   #mb_query.mode := #mb_query.c.mode.write;
   #mb_query(data_addr := 40060, data_ptr := #setting);

   "mb_station_block_footer"(sb := #sb, mb_query := #mb_query);

   (*
   Setting:

   value[1] and value[2]
   ------------------
   2 = Pascal (Pa)
   3 = kiloPascal (kPa)
   4 = megaPascal (MPa)
   5 = pounds per square inch (psi)
   6 = inches of water at 68 F
   7 = ftH2O
   8 = atm
   9 = bar
   10 = kg/cm2
   11 = g/cm2
   12 = cmHg
   13 = mmHg
   14 = torr
   15 = mH2O
   16 = cmH2O
   17 = mmH2O
   18 = inHg
   19 = mbar


   value[3]
   ------------------
   20 = degrees Celsius (ï‚°C)
   21 = degrees Fahrenheit (ï‚°F)
   22 = degrees Kelvin (K)
   23 = degrees Rankine(R)

   *)
END_FUNCTION_BLOCK

FUNCTION_BLOCK "Schneider_conzerv_EM6430"   // FB91, SCL
{ S7_Optimized_Access := 'TRUE' }
VERSION : 0.1
   VAR_INPUT
      mb_addr : USInt;
   END_VAR
   VAR_IN_OUT
      mb_query : "mb_query";
   END_VAR
   VAR
      sb : "mb_station_block_udt";
      read1_common : Struct
         Apparent_power_total : Real;
         Active_power_total : Real;
         Reactive_power_total : Real;
         Power_factor_average : Real;
         Voltage_average_phase_phase : Real;
         Voltage_average_phase_neutral : Real;
         Current_average : Real;
         Frequency : Real;   // Hz
      END_STRUCT;
      read2_phase : Array[1..3] of Struct
         Apparent_power : Real;
         Active_power : Real;
         Reactive_power : Real;
         Power_factor : Real;
         Voltage_phase_phase : Real;
         Voltage_phase_neutral : Real;
         Current : Real;
      END_STRUCT;
      read3_THD : Struct
         Voltage_THD : Array[1..3] of Real;
         Current_THD : Array[1..3] of Real;
      END_STRUCT;
      read4 : Struct
         Forward_apparent_energy : Real;
         Forward_active_energy : Real;
         Forward_reactive_inductive_energy : Real;
         Forward_reactive_capacitive_energy : Real;
         Reverse_apparent_energy : Real;
         Reverse_active_energy : Real;
         Reverse_reactive_inductive_Energy : Real;
         Reverse_reactive_capacitive_Energy : Real;
         Average_load_percentage : Real;
         Percentage_of_phase_load : Array[1..3] of Real;
         "Unbalanced_%load" : Real;
         "Unbalanced_%_voltage" : Real;
      END_STRUCT;
      read5_common_RMS : Struct
         Apparent_power_total : Real;
         Active_power_total : Real;
         Reactive_power_total : Real;
         Power_factor_average : Real;
         Voltage_average_phase_phase : Real;
         Voltage_average_phase_neutral : Real;
         Current_average : Real;
         Frequency : Real;   // Hz
         _ : UDInt;   // Reserved
         Number_of_interruption : UDInt;
      END_STRUCT;
   END_VAR
BEGIN
   // Schneider-electric - Conzerv EM6430 - Power meters
   // NHA12535-03
   // 
   // https://www.schneider-electric.com/resources/sites/SCHNEIDER_ELECTRIC/
   // content/live/FAQS/276000/FA276938/en_US/EM6430_User_Manual_NHA12535-03.pdf

   "mb_station_block_header"(sb := #sb, mb_query := #mb_query);
   #mb_query.mb_addr := #mb_addr; // Device address.

   #mb_query.mode := #mb_query.c.read.holding_reg;
   #mb_query(data_addr := 3901, data_ptr := #read1_common);
   #mb_query(data_addr := 3917, data_ptr := #read2_phase);
   #mb_query(data_addr := 3861, data_ptr := #read3_THD);
   #mb_query(data_addr := 3959, data_ptr := #read4);
   #mb_query(data_addr := 3001, data_ptr := #read5_common_RMS);

   "mb_station_block_footer"(sb := #sb, mb_query := #mb_query);
END_FUNCTION_BLOCK

// folder: Library/Modbus/Station blocks/sb Untested/S/Schneider/Altivar

FUNCTION_BLOCK "Schneider_Altivar_21_simple"   // FB123, SCL
{ S7_Optimized_Access := 'TRUE' }
VERSION : 0.1
   VAR_INPUT
      mb_addr : UInt;
      ref : Real;   // Percent
   END_VAR
   VAR_OUTPUT
      Output_frequency : Real;
   END_VAR
   VAR_IN_OUT
      mb_query : "mb_query";
   END_VAR
   VAR
      sb : "mb_station_block_udt";
      read : Struct   // 16#fd00
         frequency : Word;
         stat : Struct
            x08 : Bool;
            x09_Reverse : Bool;
            x10_Run : Bool;
            x11_Coast_stop : Bool;
            x12_Emergency_stop : Bool;
            x13_Standby_ST_ON : Bool;   // Standby: Initialization completed, not failure stop status, not alarm stop status (MOFF, LL forced stop or forced stop due to a momentary power failure), ST=ON, and RUN=ON
            x14_Standby : Bool;   // Standby: Initialization completed, not failure stop status, and not alarm stop status (MOFF, LL forced stop or forced stop due to a momentary power failure)
            x15_Local : Bool;
            x00_Failure_FL : Bool;
            x01_Failure : Bool;
            x02_Alarm : Bool;
            x03_Main_circuit_undervoltage : Bool;
            x04_THR_2 : Bool;   // THR1: PT=set value, vL, vb, Thr - THR2: PT=0, F170, F172, F173
            x05_PI_control_OFF : Bool;
            x06_Acceleration2_deceleration2 : Bool;
            x07_DC_braking : Bool;
         END_STRUCT;
      END_STRUCT;
      write : Struct
         cmd : Struct
            x08 : Bool;   // [08]
            reverse : Bool;   // [09]
            run : Bool;   // [10]
            coast_stop : Bool;   // [11]
            emergency_stop : Bool;   // [12]
            fault_reset : Bool;   // [13]
            setpoint_priority : Bool := TRUE;   // [14] Enabled regardless of the setting of FMOD
            command_priority : Bool := TRUE;   // [15] Enabled regardless of the setting of CMOD
            preset_speed_b0 : Bool;   // [00]
            preset_speed_b1 : Bool;   // [01]
            preset_speed_b2 : Bool;   // [02]
            x03 : Bool;   // [03]
            thr2 : Bool;   // [04] THR1 : PT=set value, vL, vb, tHr - THR2 : PT=0, F170, F172, F173
            PI_control : Bool;   // [05] 0:Normal operation, 1:PI OFF
            acceleration_deceleration_pattern_2 : Bool;   // [06] 0: Acceleration deceleration pattern 1
            DC_braking : Bool;   // [07]
         END_STRUCT;
         ref_speed : UInt;
      END_STRUCT;
   END_VAR
BEGIN
   // Schneider (Telemecanique) - Altivar 21 inverter
   // VFD (AC-drive)

   (*
   Param:  Name:             Default:    Options:          
   F800    Baud rate         19200       0: 9600 bps, 1: 19200 bps     
   F801    Parity            Even        0: None, 1: Even, 2: Odd      
   F802    Modbus address    1           0 ... 247                     

   CMOD    2 -> Serial communication
   FMOD    4 -> Serial communication
   *)

   "mb_station_block_header"(sb := #sb, mb_query := #mb_query);
   #mb_query.mb_addr := #mb_addr;

   #write.ref_speed := REAL_TO_UINT(#ref * 100);
   #write.cmd.run := #ref <> 0;
   #mb_query(mode := #mb_query.c.write.holding_reg,
             data_addr := 16#fa00,
             data_ptr := #write);

   // Basic data, status word.
   #mb_query(mode := #mb_query.c.read.holding_reg,
             data_addr := 16#fd00,
             data_ptr := #read);
   #Output_frequency := UINT_TO_REAL(#read.frequency) / 100; // [%]

   "mb_station_block_footer"(sb := #sb, mb_query := #mb_query);
END_FUNCTION_BLOCK

// folder: Library/Modbus/Station blocks/sb Untested/S/Schneider/Altivar/Advanced

FUNCTION_BLOCK "Schneider_Altivar_21"   // FB95, SCL
{ S7_Optimized_Access := 'TRUE' }
VERSION : 0.1
   VAR_INPUT
      mb_addr : UInt;
      ref : Real;
      acceleration_time : Real;
   END_VAR
   VAR_IN_OUT
      mb_query : "mb_query";
   END_VAR
   VAR
      sb : "mb_station_block_udt";
      data6 : Struct
         Output_current : Real;
         Voltage_DC_bus : Real;
         Output_frequency : Real;
      END_STRUCT;
      read1 : Struct   // 16#fd00
         Output_frequency : Word;
         stat : Struct
            x08 : Bool;
            x09_Reverse : Bool;
            x10_Run : Bool;
            x11_Coast_stop : Bool;
            x12_Emergency_stop : Bool;
            x13_Standby_ST_ON : Bool;   // Standby: Initialization completed, not failure stop status, not alarm stop status (MOFF, LL forced stop or forced stop due to a momentary power failure), ST=ON, and RUN=ON
            x14_Standby : Bool;   // Standby: Initialization completed, not failure stop status, and not alarm stop status (MOFF, LL forced stop or forced stop due to a momentary power failure)
            x15_Local : Bool;
            x00_Failure_FL : Bool;
            x01_Failure : Bool;
            x02_Alarm : Bool;
            x03_Main_circuit_undervoltage : Bool;
            x04_THR_2 : Bool;   // THR1: PT=set value, vL, vb, Thr - THR2: PT=0, F170, F172, F173
            x05_PI_control_OFF : Bool;
            x06_Acceleration2_deceleration2 : Bool;
            x07_DC_braking : Bool;
         END_STRUCT;
      END_STRUCT;
      read2 : Struct   // 16#fe45
         Command_mode : UInt;   // 0:Terminal board, 1:Operation panel, 2:Serial
         Setpoint_mode : UInt;   // 1 VIA, 2 VIB, 3 Operation panel, 4 Serial, 5 TB up down frequency, 255 Preset speed operation
      END_STRUCT;
      read3_alarm : Struct   // 16#fe91
         x08_Over_torque : Bool;
         x09_Cumulative_operation_hours : Bool;
         x10 : Bool;
         x11 : Bool;
         x12 : Bool;
         "x13_Main circuit_undervoltage" : Bool;   // same as MS-relay status
         x14_Decelerating_stopping : Bool;   // Related: F256 setting. At the time of the instant blackout, Forced deceleration/stop
         x15_Decelerating_stopping : Bool;   // Related: F302 setting. An automatic stop during the lower limit frequency continuance
         x00_Overcurrent : Bool;
         x01_Inverter_overload : Bool;
         x02_Motor_overload : Bool;
         x03_Overheat : Bool;
         x04_Overvoltage : Bool;
         x05_Main_circuit_undervoltage : Bool;
         x06 : Bool;
         x07_Undercurrent : Bool;
      END_STRUCT;
      read4_alarm2 : Struct   // 16#fe79
         x08 : Bool;
         x09 : Bool;
         x10 : Bool;
         x11 : Bool;
         x12 : Bool;
         x13 : Bool;
         x14 : Bool;
         x15 : Bool;
         x00_Fan_life_alarm : Bool;
         x01_Circuit_board_life : Bool;
         x02_Main_circuit_capacitor_life : Bool;
         x03_User_set_alarm : Bool;
         x04 : Bool;
         x05 : Bool;
         x06 : Bool;
         x07 : Bool;
      END_STRUCT;
      read5_trip_code : UInt;   // 16#fc90
      write1 : Struct
         cmd : Struct
            x08 : Bool;   // [08]
            reverse : Bool;   // [09]
            run : Bool;   // [10]
            coast_stop : Bool;   // [11]
            emergency_stop : Bool;   // [12]
            fault_reset : Bool;   // [13]
            setpoint_priority : Bool := TRUE;   // [14] Enabled regardless of the setting of FMOD
            command_priority : Bool := TRUE;   // [15] Enabled regardless of the setting of CMOD
            preset_speed_b0 : Bool;   // [00]
            preset_speed_b1 : Bool;   // [01]
            preset_speed_b2 : Bool;   // [02]
            x03 : Bool;   // [03]
            thr2 : Bool;   // [04] THR1 : PT=set value, vL, vb, tHr - THR2 : PT=0, F170, F172, F173
            PI_control : Bool;   // [05] 0:Normal operation, 1:PI OFF
            acceleration_deceleration_pattern_2 : Bool;   // [06] 0: Acceleration deceleration pattern 1
            DC_braking : Bool;   // [07]
         END_STRUCT;
         ref : UInt;
      END_STRUCT;
      write2_comm_fault_action : UInt;
      _ : Bool;
      sequence : "mb_sequence";
   END_VAR
   VAR_TEMP
      read6 : Struct   // 16#fe03
         Output_current : UInt;
         Voltage_DC_bus : UInt;
      END_STRUCT;
      u : UInt;
   END_VAR
BEGIN
   // Schneider (Telemecanique) - Altivar 21 inverter
   // VFD (AC-drive)

   (*
   Param:  Name:             Default:    Options:          
   F800    Baud rate         19200       0: 9600 bps, 1: 19200 bps     
   F801    Parity            Even        0: None, 1: Even, 2: Odd      
   F802    Modbus address    1           0 ... 247                     

   CMOD    2 -> Serial communication
   FMOD    4 -> Serial communication
   *)

   "mb_station_block_header"(sb := #sb, mb_query := #mb_query);
   #mb_query.mb_addr := #mb_addr;

   REGION Low priority queries     
       #sequence.conf.first_state := 1600;
       CASE "mb_sequence_init"(sequence := #sequence, mb_query := #mb_query) OF
               // ----- READ HOLDING REG ----- (State 3xx)
           300: // Where the drive take commands from: modbus or Terminal board.
               #mb_query(data_addr := 16#fe45, data_ptr := #read2); // 65093
           301: #mb_query(data_addr := 16#fe91, data_ptr := #read3_alarm);
           302: #mb_query(data_addr := 16#fe79, data_ptr := #read4_alarm2);
           303: #mb_query(data_addr := 16#fc90, data_ptr := #read5_trip_code);
           304: // Other data: Current, DC-bus
               #mb_query(data_addr := 16#fe03, data_ptr := #read6);
               IF #mb_query.Done THEN
                   #data6.Output_current := UINT_TO_REAL(#read6.Output_current) / 100;
                   #data6.Voltage_DC_bus := UINT_TO_REAL(#read6.Voltage_DC_bus) / 100;
               END_IF;
               #sequence.next_state := 1600;

               // ----- WRITE MULTIPLE HOLDING REG ----- (State 16xx)
           1600: // Behaviour on modbus fault
               #mb_query(data_addr := 16#f603, data_ptr := #write2_comm_fault_action);
           1601: // Acceleration time 1  (0.1)
               #u := REAL_TO_UINT(#acceleration_time * 10);
               #mb_query(data_addr := 16#f603, data_ptr := #u);
               #sequence.next_state := 300;
           ELSE
               #sequence.state += 1;
       END_CASE;
       #sequence(sb := #sb, mb_query := #mb_query);
   END_REGION

   REGION High priotiry querie     
       #write1.ref := REAL_TO_UINT(#ref * 100);
       #write1.cmd.run := #ref <> 0 AND #sequence.Done;
       #mb_query(mode := #mb_query.c.write.holding_reg, // 64000
                 data_addr := 16#fa00,
                 data_ptr := #write1);

       // Basic data, status word.
       #mb_query(mode := #mb_query.c.read.holding_reg,
                 data_addr := 16#fd00,
                 data_ptr := #read1); // 64768
       IF #mb_query.Done THEN
           #data6.Output_frequency :=
           (* *)UINT_TO_REAL(#read1.Output_frequency) / 100; // [%]
       END_IF;
   END_REGION

   "mb_station_block_footer"(sb := #sb, mb_query := #mb_query);

   (* Trip codes:
   NErr     0  0  No error
   OC1      1  1  Over-current during acceleration
   OC2      2  2  Over-current during deceleration
   OC3      3  3  Over-current during constant speed operation
   OCL      4  4  Over-current in load at startup
   OCA      5  5  Short circuit in arm
   EPHI     8  8  Input phase failure
   EPHO     9  9  Output phase failure
   OP1      A 10 Overvoltage during acceleration
   OP2      B 11 Overvoltage during deceleration
   OP3      C 12 Overvoltage during constant speed operation
   OL1      D 13 Over-LOAD in inverter
   OL2      E 14 Over-LOAD in motor
   OH      10 16 Overheat trip
   E       11 17 Emergency stop
   EEP1    12 18 EEPROM fault 1 (writing error)
   EEP2    13 19 EEPROM fault 2 (reading error)
   EEP3    14 20 EEPROM fault 3 (internal fault)
   Err2    15 21 RAM fault
   Err3    16 22 ROM fault
   Err4    17 23 CPU fault
   Err5    18 24 Communication error trip
   Err7    1A 26 Current detector fault
   Err8    1B 27 Optional circuit board type error
   UC      1D 29 Small-current trip
   UP1     1E 30 Trip due to undervoltage in main circuit
   Ot      20 32 Over-torque trip
   EF2     22 34 Ground fault trip (hardware detection)
   OC1P    25 37 Overcurrent flowing in element during acceleration
   OC2P    26 38 Overcurrent flowing in element during deceleration
   OC3P    27 39 Overcurrent flowing in element during operation
   EtYP    29 41 Inverter type error
   OH2     2E 46 External thermal input
   SOUt    2F 47 VIA cable break
   E-18    32 50 Break in an analog signal cable
   E-19    33 51 CPU fault
   E-20    34 52 Excess torque boost
   E-21    35 53 CPU fault
   Etn1    54 84 Auto-tuning error
   *)
END_FUNCTION_BLOCK

// folder: Library/Modbus/Station blocks/sb Untested/S/Schneider/Power meters

FUNCTION_BLOCK "Schneider_power_meter"   // FB2, SCL
{ S7_Optimized_Access := 'TRUE' }
VERSION : 0.1
   VAR_INPUT
      mb_addr : USInt;
   END_VAR
   VAR_IN_OUT
      mb_query : "mb_query";
   END_VAR
   VAR RETAIN
      conf : Struct
         power_system : UInt := 65535;   // 0=1PH2W L–N, 1=1PH2W L–L, 2=1PH3W L–L with N, 3=3PH3W, 11=3PH4W, 13=1PH4W multi-L with N
      END_STRUCT;
   END_VAR
   VAR
      sb : "mb_station_block_udt";
      "e" : Int;   // Error
      data : "energy_udt";
      frequency : Real;
      temperature : Real;
      serial_number : UDInt;
      power_factor : Struct
         L : Array[1..3] of Real;
         total : Real;
         displacement : Struct
            L : Array[1..3] of Real;
            total : Real;
         END_STRUCT;
      END_STRUCT;
      unbalanced : Struct
         current : Struct
            L : Array[1..3] of Real;
            worst : Real;
         END_STRUCT;
         voltage : Struct
            L_L : Array[1..3] of Real;
            L_L_worst : Real;
            L_N : Array[1..3] of Real;
            L_N_worst : Real;
         END_STRUCT;
      END_STRUCT;
      tangent_phi : Real;
      tmp : DWord;
   END_VAR
   VAR CONSTANT
      ALL : DInt := 0;
   END_VAR
BEGIN
   // Schneider - PowerLogic  (Power meter)
   // PM3200, PM3210, PM3250, PM3255, PM5560, PM5563, PM5563RD
   //
   // DOCA0006EN-06  -  08/2016
   // Default com.: 19200/8-E-1. Default addr: 1
   // 
   // https://www.se.com/ww/en/product/METSEPM3250/pm3250-power-meter---rs485/
   // https://download.schneider-electric.com/files?p_enDocType=User+guide&p_File_Name=DOCA0006EN-06.pdf&p_Doc_Ref=DOCA0006EN
   // https://www.schneider-electric.com/en/faqs/FA234017/
   //
   // Apparently there is a error in the datasheet, all register
   // addresses are added by two. Eg 3000 is actually 2998.

   "mb_station_block_header"(sb := #sb, mb_query := #mb_query );
   #mb_query.mb_addr := #mb_addr;
   #mb_query.mode := #mb_query.c.read.holding_reg;

   IF "mb_query_range"(start := 128, end := 129, q := #mb_query) THEN
       #"e" += "mb_swap_word"(start := #ALL, end := #ALL,  q := #mb_query);
       #"e" += "mb_read_buffer"(addr := 130-2, ptr := #serial_number, q := #mb_query);
   END_IF;

   IF "mb_query_range"(start := 2700-2, end := 2710-1, q := #mb_query) THEN
       #"e" += "mb_swap_word"(start := #ALL, end := #ALL,  q := #mb_query);
       #"e" += "mb_read_buffer"(addr := 2700-2, ptr := #data.energy.active_out, q := #mb_query);
       #"e" += "mb_read_buffer"(addr := 2702-2, ptr := #data.energy.active_in, q := #mb_query);
       #"e" += "mb_read_buffer"(addr := 2704-2, ptr := #data.energy.reactive_out, q := #mb_query);
       #"e" += "mb_read_buffer"(addr := 2706-2, ptr := #data.energy.reactive_in, q := #mb_query);
       #"e" += "mb_read_buffer"(addr := 2708-2, ptr := #data.energy.apparent_out, q := #mb_query);
       #"e" += "mb_read_buffer"(addr := 2710-2, ptr := #data.energy.apparent_in, q := #mb_query);
   END_IF;

   IF "mb_query_range"(start := 3000-2, end := 3076-1, q := #mb_query) THEN
       #"e" += "mb_swap_word"(start := #ALL, end := #ALL,  q := #mb_query);
       #"e" += "mb_read_buffer"(addr := 3000-2, ptr := #data.current.L, q := #mb_query);
       #"e" += "mb_read_buffer"(addr := 3006-2, ptr := #data.current.N, q := #mb_query);
       #"e" += "mb_read_buffer"(addr := 3010-2, ptr := #data.current.avg, q := #mb_query);
       #"e" += "mb_read_buffer"(addr := 3012-2, ptr := #unbalanced.current.L, q := #mb_query);
       #"e" += "mb_read_buffer"(addr := 3018-2, ptr := #unbalanced.current.worst, q := #mb_query);
       #"e" += "mb_read_buffer"(addr := 3020-2, ptr := #data.voltage.L_L, q := #mb_query);
       #"e" += "mb_read_buffer"(addr := 3026-2, ptr := #data.voltage.L_L_avg, q := #mb_query);
       #"e" += "mb_read_buffer"(addr := 3028-2, ptr := #data.voltage.L_N, q := #mb_query);
       #"e" += "mb_read_buffer"(addr := 3036-2, ptr := #data.voltage.L_N_avg, q := #mb_query);
       #"e" += "mb_read_buffer"(addr := 3038-2, ptr := #unbalanced.voltage.L_L, q := #mb_query);
       #"e" += "mb_read_buffer"(addr := 3044-2, ptr := #unbalanced.voltage.L_L_worst, q := #mb_query);
       #"e" += "mb_read_buffer"(addr := 3046-2, ptr := #unbalanced.voltage.L_N, q := #mb_query);
       #"e" += "mb_read_buffer"(addr := 3052-2, ptr := #unbalanced.voltage.L_N_worst, q := #mb_query);
       #"e" += "mb_read_buffer"(addr := 3054-2, ptr := #data.power.active, q := #mb_query);
       #"e" += "mb_read_buffer"(addr := 3060-2, ptr := #data.power.active.total, q := #mb_query);
       #"e" += "mb_read_buffer"(addr := 3062-2, ptr := #data.power.reactive, q := #mb_query);
       #"e" += "mb_read_buffer"(addr := 3068-2, ptr := #data.power.reactive.total, q := #mb_query);
       #"e" += "mb_read_buffer"(addr := 3070-2, ptr := #data.power.apparent, q := #mb_query);
       #"e" += "mb_read_buffer"(addr := 3076-2, ptr := #data.power.apparent.total, q := #mb_query);
   END_IF;

   IF "mb_query_range"(start := 3078-2, end := 3084-1, q := #mb_query) THEN
       #"e" += "mb_swap_word"(start := #ALL, end := #ALL,  q := #mb_query);
       #"e" += "mb_read_buffer"(addr := 3078-2, ptr := #power_factor.L, q := #mb_query);
       #"e" += "mb_read_buffer"(addr := 3084-2, ptr := #power_factor.total, q := #mb_query);
       #"e" += "mb_read_buffer"(addr := 3084-2, ptr := #power_factor.displacement, q := #mb_query);
   END_IF;

   IF "mb_query_range"(start := 3108-2, end := 3132-1, q := #mb_query) THEN
       #"e" += "mb_swap_word"(start := #ALL, end := #ALL,  q := #mb_query);
       #"e" += "mb_read_buffer"(addr := 3108-2, ptr := #tangent_phi, q := #mb_query);
       #"e" += "mb_read_buffer"(addr := 3110-2, ptr := #frequency, q := #mb_query);
       #"e" += "mb_read_buffer"(addr := 3132-2, ptr := #temperature, q := #mb_query);
   END_IF;


   // ---------------------- WRITE HOLDING REGISTER QURIES ---------------------- 
   #mb_query.mode := #mb_query.c.write.holding_reg;

   IF #conf.power_system <> 65535 THEN
       #mb_query(data_addr := 2016, data_ptr := #conf.power_system);
   END_IF; 


   "mb_station_block_footer"(sb := #sb, mb_query := #mb_query );

   (* 
   Power factor:
   -2 < PF < -1: Quad 2, active power negative, capacitive
   -1 < PF <  0: Quad 3, active power negative, inductive
    0 < PF <  1: Quad 1, active power positive, inductive
    1 < PF <  2: Quad 4, active power positive, capacitive     

   #conf.power_system :
   0 = 1PH2W L–N
   1 = 1PH2W L–L
   2 = 1PH3W L–L with N
   3 = 3PH3W
   11 = 3PH4W
   13 = 1PH4W multi-L with N      


   *)
END_FUNCTION_BLOCK

FUNCTION_BLOCK "Schneider_PM1000_series"   // FB49, SCL
TITLE = Schneider Electric - PM1000 Series Power Meters
{ S7_Optimized_Access := 'TRUE' }
VERSION : 0.1
   VAR_INPUT
      mb_addr : UInt;
   END_VAR
   VAR_OUTPUT
      all : Struct
         apparent_power : Real;
         active_power : Real;
         reactive_power : Real;
         power_factor : Real;
         voltage_L_L : Real;
         voltage_L_N : Real;
         current : Real;
      END_STRUCT;
      phase : Array[1..3] of Struct
         apparent_power : Real;
         active_power : Real;
         reactive_power : Real;
         power_factor : Real;
         voltage_L_L : Real;
         voltage_L_N : Real;
         current : Real;
      END_STRUCT;
   END_VAR
   VAR_IN_OUT
      mb_query : "mb_query";
   END_VAR
   VAR
      sb : "mb_station_block_udt";
   END_VAR
   VAR_TEMP
      tAll : Struct
         apparent_power : DWord;
         active_power : DWord;
         reactive_power : DWord;
         power_factor : DWord;
         voltage_L_L : DWord;
         voltage_L_N : DWord;
         current : DWord;
      END_STRUCT;
      tPhase : Array[1..3] of Struct
         apparent_power : DWord;
         active_power : DWord;
         reactive_power : DWord;
         power_factor : DWord;
         voltage_L_L : DWord;
         voltage_L_N : DWord;
         current : DWord;
      END_STRUCT;
      c : Int;
   END_VAR
BEGIN
   // Schneider Electric - PowerLogic - PM1000 Series Power Meters
   //  - PM1200
   // 
   // http://static.schneider-electric.us/docs/Power%20Management/
   // PowerLogic%20Products/Metering/PM1200%20power%20meter/
   // PLSED309039EN_PM1000_UG.pdf

   "mb_station_block_header"(sb := #sb,
                             mb_query := #mb_query);
   #mb_query.mb_addr := #mb_addr;

   #mb_query.mode := #mb_query.c.read.holding_reg;

   #mb_query(data_addr := 3901,
             data_ptr := #tAll);
   IF #mb_query.Done THEN
       #all.apparent_power := DWORD_TO_REAL(SWAP(#tAll.apparent_power));
       #all.active_power := DWORD_TO_REAL(SWAP(#tAll.active_power));
       #all.reactive_power := DWORD_TO_REAL(SWAP(#tAll.reactive_power));
       #all.power_factor := DWORD_TO_REAL(SWAP(#tAll.power_factor));
       #all.voltage_L_L := DWORD_TO_REAL(SWAP(#tAll.voltage_L_L));
       #all.voltage_L_N := DWORD_TO_REAL(SWAP(#tAll.voltage_L_N));
       #all.current := DWORD_TO_REAL(SWAP(#tAll.current));
   END_IF;

   FOR #c := 1 TO 3 DO
       CASE #c OF
           1:
               #mb_query.data_addr := 3917;
           2:
               #mb_query.data_addr := 3931;
           3:
               #mb_query.data_addr := 3945;
       END_CASE;
       #mb_query(data_ptr := #tPhase[#c]);
       IF #mb_query.Done THEN
           #phase[#c].apparent_power := DWORD_TO_REAL(SWAP(#tPhase[#c].apparent_power));
           #phase[#c].active_power := DWORD_TO_REAL(SWAP(#tPhase[#c].active_power));
           #phase[#c].reactive_power := DWORD_TO_REAL(SWAP(#tPhase[#c].reactive_power));
           #phase[#c].power_factor := DWORD_TO_REAL(SWAP(#tPhase[#c].power_factor));
           #phase[#c].voltage_L_L := DWORD_TO_REAL(SWAP(#tPhase[#c].voltage_L_L));
           #phase[#c].voltage_L_N := DWORD_TO_REAL(SWAP(#tPhase[#c].voltage_L_N));
           #phase[#c].current := DWORD_TO_REAL(SWAP(#tPhase[#c].current));
       END_IF;
   END_FOR;

   "mb_station_block_footer"(sb := #sb,
                             mb_query := #mb_query);
END_FUNCTION_BLOCK

FUNCTION_BLOCK "Schneider_PM750"   // FB92, SCL
{ S7_Optimized_Access := 'TRUE' }
VERSION : 0.1
   VAR_INPUT
      mb_addr : UInt;
   END_VAR
   VAR_IN_OUT
      mb_query : "mb_query";
   END_VAR
   VAR
      sb : "mb_station_block_udt";
      data1 : Struct
         "Real Energy, Total" : Real;   // kWh
         "Apparent Energy,Tota" : Real;   // kVAh
         "Reactive Energy,Tota" : Real;   // kVARh
         "Real Power, Total" : Real;   // kW
         "Apparent Power, Total" : Real;   // kVA
         "Reactive Power, Total" : Real;   // kVAR
         "Power Factor, Total" : Real;
         "Voltage, L-L, 3PAverage" : Real;   // Volt
         "Voltage, L-N, 3PAverage" : Real;   // Volt
         "Current, 3P Average" : Real;   // Amp
         Frequency : Real;
      END_STRUCT;
      data2 : Struct
         Current : Array[1..3] of Real;
         Current_N : Real;
      END_STRUCT;
      data3 : Struct
         Voltage_L_L : Array[1..3] of Real;   // [V] 1:L1-L2, 2:L2-L3, 3:L3-L1
         Voltage_L_N : Array[1..3] of Real;   // [V]
         "Real Power" : Array[1..3] of Real;   // kW
         "Apparent Power" : Array[1..3] of Real;   // kVA
         "Reactive Power" : Array[1..3] of Real;   // kVAR
      END_STRUCT;
   END_VAR
BEGIN
   // Schneider - Power Meter 750
   // 63230-507-201A1 - 03/2007
   // 
   // Web: https://www.ccontrols.com/support/dp/SchneiderElectricPowerMeter750.pdf

   "mb_station_block_header"(sb := #sb, mb_query := #mb_query);
   #mb_query.mb_addr := #mb_addr;

   #mb_query.mode := #mb_query.c.read.holding_reg;
   #mb_query(data_addr := 1000, data_ptr := #data1);
   #mb_query(data_addr := 1034, data_ptr := #data2);
   #mb_query(data_addr := 1054, data_ptr := #data3);

   "mb_station_block_footer"(sb := #sb, mb_query := #mb_query);
END_FUNCTION_BLOCK

// folder: Library/Modbus/Station blocks/sb Untested/S/Schneider/Power meters/z Deprecated

FUNCTION_BLOCK "Schneider_PM556x_series"   // FB48, SCL
{ S7_Optimized_Access := 'TRUE' }
VERSION : 0.1
   VAR_INPUT
      mb_addr : UInt;
   END_VAR
   VAR_IN_OUT
      mb_query : "mb_query";
   END_VAR
   VAR
      sb : "mb_station_block_udt";
      Accumulated_Energy : Struct
         "Active Energy Delivered (Into Load)" : Real;   // kWh
         "Active Energy Received (Out of Load)" : Real;   // kWh
         "Active Energy Delivered + Received" : Real;   // kWh
         "Active Energy Delivered- Received" : Real;   // kWh
         "Reactive Energy Delivered" : Real;   // kVARh
         "Reactive Energy Received" : Real;   // kVARh
         "Reactive Energy Delivered + Received" : Real;   // kVARh
         "Reactive Energy Delivered - Received" : Real;   // kVARh
         "Apparent Energy Delivered" : Real;   // kVAh
         "Apparent Energy Received" : Real;   // kVAh
         "Apparent Energy Delivered + Received" : Real;   // kVAh
         "Apparent Energy Delivered - Received" : Real;   // kVAh
      END_STRUCT;
      data1 : Struct
         Current : Array[1..3] of Real;   // A
         "Current N" : Real;   // A
         "Current G" : Real;   // A
         "Current Avg" : Real;   // A
         "Current Unbalance" : Array[1..3] of Real;   // %
         "Current Unbalance Worst" : Real;   // %
         "Voltage L-L" : Array[1..3] of Real;   // V
         "Voltage L-L Avg" : Real;   // V
         "Voltage L-N" : Array[1..3] of Real;   // V
         "Voltage L-N Avg" : Real;   // V
         "Voltage Unbalance L-L" : Array[1..3] of Real;   // %
         "Voltage Unbalance L-L Worst" : Real;   // %
         "Voltage Unbalance L-N" : Array[1..3] of Real;   // %
         "Voltage Unbalance L-N Worst" : Real;   // %
      END_STRUCT;
      Power : Struct
         "Active Power" : Array[1..3] of Real;   // kW
         "Active Power Total" : Real;   // kW
         "Reactive Power" : Array[1..3] of Real;   // kVAR
         "Reactive Power Total" : Real;   // kVAR
         "Apparent Power" : Array[1..3] of Real;   // kVA
         "Apparent Power Total" : Real;   // kVA
         "Power Factor" : Array[1..3] of Real;   // ---
         "Power Factor Total" : Real;   // ---
         "Displacement Power Factor" : Array[1..3] of Real;   // ---
         "Displacement Power Factor Total" : Real;   // ---
      END_STRUCT;
      PF : Struct
         "Power Factor" : Array[1..3] of Real;
         "Power Factor Total" : Real;
         "Displacement Power Factor" : Array[1..3] of Real;
         "Displacement Power Factor Total" : Real;
      END_STRUCT;
      Frequency : Real;   // Hz
   END_VAR
   VAR_TEMP
      c : Int;
      t1 : Real;
      t2 : Real;
   END_VAR
BEGIN
   // Schneider Electric - PM5560, PM5563, PM5563RD
   // 
   // https://www.schneider-electric.com/en/faqs/FA234017/

   "mb_station_block_header"(sb := #sb, mb_query := #mb_query);
   #mb_query.mb_addr := #mb_addr;

   #mb_query.mode := #mb_query.c.read.holding_reg;
   #mb_query(data_addr := 2700, data_ptr := #Accumulated_Energy);
   #mb_query(data_addr := 3000, data_ptr := #data1);
   #mb_query(data_addr := 3054, data_ptr := #Power);
   #mb_query(data_addr := 3110, data_ptr := #Frequency);

   "mb_station_block_footer"(sb := #sb, mb_query := #mb_query);

   FOR #c := 1 TO 8 DO
       (* Power factor values are specially encoded floating point 
       values. Angle of complex power = power factor register value
       0° = 1, 90° = 0,  180° = -1,  270° = 2,  Q1: 0 < x < 1
       Q2: -2 < x < -1,  Q3:  -1 < x < 0,   Q4: 1 < x < 2  *)
       CASE #c OF
           1..3: #t1 := #Power."Power Factor"[#c];
           4:    #t1 := #Power."Power Factor Total";
           5..7: #t1 := #Power."Displacement Power Factor"[#c - 4];
           8:    #t1 := #Power."Displacement Power Factor Total";
       END_CASE;
       IF #t1 > 1 THEN // PF is leading
           #t2 := 2 - #t1;
       ELSIF #t1 < -1 THEN // PF is leading
           #t2 := -2 - #t1;
       ELSE            // ABS(#t1) = 1 -> PF is at unity
           #t2 := #t1; // else -> PF is lagging
       END_IF;
       CASE #c OF
           1..3: #PF."Power Factor"[#c] := #t2;
           4:    #PF."Power Factor Total" := #t2;
           5..7: #PF."Displacement Power Factor"[#c - 4] := #t2;
           8:    #PF."Displacement Power Factor Total" := #t2;
       END_CASE;
   END_FOR;
END_FUNCTION_BLOCK

FUNCTION_BLOCK "Schneider_power_meter_750"   // FB50, SCL
{ S7_Optimized_Access := 'TRUE' }
VERSION : 0.1
   VAR_INPUT
      mb_addr : UInt;
   END_VAR
   VAR_IN_OUT
      mb_query : "mb_query";
   END_VAR
   VAR
      sb : "mb_station_block_udt";
      data1 : Struct
         "Real Energy, Total" : Real;   // kWh
         "Apparent Energy,Tota" : Real;   // kVAh
         "Reactive Energy,Tota" : Real;   // kVARh
         "Real Power, Total" : Real;   // kW
         "Apparent Power, Total" : Real;   // kVA
         "Reactive Power, Total" : Real;   // kVAR
         "Power Factor, Total" : Real;
         "Voltage, L-L, 3PAverage" : Real;   // Volt
         "Voltage, L-N, 3PAverage" : Real;   // Volt
         "Current, 3P Average" : Real;   // Amp
         Frequency : Real;
      END_STRUCT;
      data2 : Struct
         Current : Array[1..3] of Real;
         Current_N : Real;
      END_STRUCT;
      data3 : Struct
         Voltage_L_L : Array[1..3] of Real;   // [V] 1:L1-L2, 2:L2-L3, 3:L3-L1
         Voltage_L_N : Array[1..3] of Real;   // [V]
         "Real Power" : Array[1..3] of Real;   // kW
         "Apparent Power" : Array[1..3] of Real;   // kVA
         "Reactive Power" : Array[1..3] of Real;   // kVAR
      END_STRUCT;
   END_VAR
BEGIN
   // Schneider - Power Meter 750
   // 63230-507-201A1 - 03/2007
   // 
   // Web: https://www.ccontrols.com/support/dp/SchneiderElectricPowerMeter750.pdf

   "mb_station_block_header"(sb := #sb,
                             mb_query := #mb_query);
   #mb_query.mb_addr := #mb_addr;

   #mb_query.mode := #mb_query.c.read.holding_reg;
   #mb_query(data_addr := 1000,
             data_ptr := #data1);
   #mb_query(data_addr := 1034,
             data_ptr := #data2);
   #mb_query(data_addr := 1054,
             data_ptr := #data3);

   "mb_station_block_footer"(sb := #sb,
                             mb_query := #mb_query);
END_FUNCTION_BLOCK

// folder: Library/Modbus/Station blocks/sb Untested/S/Siemens

FUNCTION_BLOCK "Siemens_7SR11_7SR12_argus"   // FB53, SCL
{ S7_Optimized_Access := 'TRUE' }
VERSION : 0.1
   VAR_INPUT
      mb_addr : USInt := 1;
   END_VAR
   VAR_OUTPUT
      out1 : Struct
         primary_Voltage_L_L : Array[1..3] of Real;
         primary_Voltage_L_N : Array[1..3] of Real;
         secondary_Voltage_L_N : Array[1..3] of Real;
      END_STRUCT;
      out2 : Struct
         nominal_voltage_degrees_L_L : Array[1..3] of Real;
         nominal_voltage_degrees_L_N : Array[1..3] of Real;
         Vzps : Real;
         Vpps : Real;
         Vnps : Real;
         Vzps_degree : Real;
         Vpps_degree : Real;
         Vnps_degree : Real;
         frequency : Real;
      END_STRUCT;
      out3 : Struct
         primary_current : Array[1..3] of Real;
         secondary_current : Array[1..3] of Real;
         nominal_current : Array[1..3] of Real;
         nominal_current_degrees : Array[1..3] of Real;
         primary_In : Real;
         secondary_In : Real;
         nominal_In : Real;
         primary_Ig : Real;
         secondary_Ig : Real;
         nominal_Ig : Real;
         nominal_Izps : Real;
         nominal_Ipps : Real;
         nominal_Inps : Real;
         nominal_Izps_degrees : Real;
         nominal_Ipps_degrees : Real;
         nominal_Inps_degrees : Real;
      END_STRUCT;
      out4 : Struct
         active_power : Array[1..3] of Real;
         active_power_tot : Real;
         reactive_power : Array[1..3] of Real;
         reactive_power_tot : Real;
         apparent_power : Array[1..3] of Real;
         apparent_power_tot : Real;
         power_factor : Array[1..3] of Real;
         power_factor_tot : Real;
      END_STRUCT;
   END_VAR
   VAR_IN_OUT
      mb_query : "mb_query";
   END_VAR
   VAR
      sb : "mb_station_block_udt";
      out5 : Struct
         act_energy_exp : UDInt;
         act_energy_imp : UDInt;
         react_energy_exp : UDInt;
         react_energy_imp : UDInt;
         thermal_status_Ph_A : UInt;
         thermal_status_Ph_B : UInt;
         thermal_Status_Ph_C : UInt;
      END_STRUCT;
      out6 : Struct
         fault_records : Real;
         event_records : Real;
         waveform_records : Real;
         secondary_voltage : Array[1..3] of Real;
      END_STRUCT;
   END_VAR
   VAR_TEMP
      c : Int;
      read1 : Struct
         primary_Voltage_L_L : Array[1..3] of UDInt;
         primary_Voltage_L_N : Array[1..3] of UDInt;
         secondary_Voltage_L_N : Array[1..3] of UDInt;
      END_STRUCT;
      read2 : Struct
         nominal_voltage_degrees_L_L : Array[1..3] of UDInt;
         nominal_voltage_degrees_L_N : Array[1..3] of UDInt;
         Vzps : UDInt;
         Vpps : UDInt;
         Vnps : UDInt;
         Vzps_degree : UDInt;
         Vpps_degree : UDInt;
         Vnps_degree : UDInt;
         frequency : UDInt;
      END_STRUCT;
      read3 : Struct
         primary_current : Array[1..3] of UDInt;
         secondary_current : Array[1..3] of UDInt;
         nominal_current : Array[1..3] of UDInt;
         nominal_current_degrees : Array[1..3] of UDInt;
         primary_In : UDInt;
         secondary_In : UDInt;
         nominal_In : UDInt;
         primary_Ig : UDInt;
         secondary_Ig : UDInt;
         nominal_Ig : UDInt;
         nominal_Izps : UDInt;
         nominal_Ipps : UDInt;
         nominal_Inps : UDInt;
         nominal_Izps_degrees : UDInt;
         nominal_Ipps_degrees : UDInt;
         nominal_Inps_degrees : UDInt;
      END_STRUCT;
      read4 : Struct
         active_power : Array[1..3] of UDInt;
         active_power_tot : UDInt;
         reactive_power : Array[1..3] of UDInt;
         reactive_power_tot : UDInt;
         apparent_power : Array[1..3] of UDInt;
         apparent_power_tot : UDInt;
         power_factor : Array[1..3] of UDInt;
         power_factor_tot : UDInt;
      END_STRUCT;
      read6 : Struct
         fault_records : UDInt;
         event_records : UDInt;
         waveform_Records : UDInt;
         secondary_voltage : Array[1..3] of UDInt;
      END_STRUCT;
   END_VAR
BEGIN
   // Siemens - 7SR11 & 7SR12 - Argus - Overcurrent Relay
   // Energy Management
   //  
   // - https://cache.industry.siemens.com/dl/files/284/109747284/
   //   att_928907/v1/7SR12_Argus_Complete_Technical_Manual.pdf
   //   ==> page 212  

   "mb_station_block_header"(sb := #sb,
                             mb_query := #mb_query);
   #mb_query.mb_addr := #mb_addr;

   #mb_query.mode := #mb_query.c.mode.read;

   #mb_query(data_addr := 40010,
             data_ptr := #read1);
   IF #mb_query.Done THEN
       FOR #c := 1 TO 3 DO
           #out1.primary_Voltage_L_L[#c] := UDINT_TO_REAL(#read1.primary_Voltage_L_L[#c]) / 1000;
           #out1.primary_Voltage_L_N[#c] := UDINT_TO_REAL(#read1.primary_Voltage_L_N[#c]) / 1000;
           #out1.secondary_Voltage_L_N[#c] := UDINT_TO_REAL(#read1.secondary_Voltage_L_N[#c]) / 1000;
       END_FOR;
   END_IF;

   #mb_query(data_addr := 40034,
             data_ptr := #read2);
   IF #mb_query.Done THEN
       FOR #c := 1 TO 3 DO
           #out2.nominal_voltage_degrees_L_L[#c] := UDINT_TO_REAL(#read2.nominal_voltage_degrees_L_L[#c]) / 1000;
           #out2.nominal_voltage_degrees_L_N[#c] := UDINT_TO_REAL(#read2.nominal_voltage_degrees_L_N[#c]) / 1000;
       END_FOR;
       #out2.Vzps := UDINT_TO_REAL(#read2.Vzps) / 1000;
       #out2.Vpps := UDINT_TO_REAL(#read2.Vpps) / 1000;
       #out2.Vnps := UDINT_TO_REAL(#read2.Vnps) / 1000;
       #out2.Vzps_degree := UDINT_TO_REAL(#read2.Vzps_degree) / 1000;
       #out2.Vpps_degree := UDINT_TO_REAL(#read2.Vpps_degree) / 1000;
       #out2.Vnps_degree := UDINT_TO_REAL(#read2.Vnps_degree) / 1000;
       #out2.frequency := UDINT_TO_REAL(#read2.frequency) / 1000;
   END_IF;

   #mb_query(data_addr := 40064,
             data_ptr := #read3);
   IF #mb_query.Done THEN
       FOR #c := 1 TO 3 DO
           #out3.primary_current[#c] := UDINT_TO_REAL(#read3.primary_current[#c]) / 1000;
           #out3.secondary_current[#c] := UDINT_TO_REAL(#read3.secondary_current[#c]) / 1000;
           #out3.nominal_current[#c] := UDINT_TO_REAL(#read3.nominal_current[#c]) / 1000;
           #out3.nominal_current_degrees[#c] := UDINT_TO_REAL(#read3.nominal_current_degrees[#c]) / 1000;
       END_FOR;
       #out3.primary_In := UDINT_TO_REAL(#read3.primary_In) / 1000;
       #out3.secondary_In := UDINT_TO_REAL(#read3.secondary_In) / 1000;
       #out3.nominal_In := UDINT_TO_REAL(#read3.nominal_In) / 1000;
       #out3.primary_Ig := UDINT_TO_REAL(#read3.primary_Ig) / 1000;
       #out3.secondary_Ig := UDINT_TO_REAL(#read3.secondary_Ig) / 1000;
       #out3.nominal_Ig := UDINT_TO_REAL(#read3.nominal_Ig) / 1000;
       #out3.nominal_Izps := UDINT_TO_REAL(#read3.nominal_Izps) / 1000;
       #out3.nominal_Ipps := UDINT_TO_REAL(#read3.nominal_Ipps) / 1000;
       #out3.nominal_Inps := UDINT_TO_REAL(#read3.nominal_Inps) / 1000;
       #out3.nominal_Izps_degrees := UDINT_TO_REAL(#read3.nominal_Izps_degrees) / 1000;
       #out3.nominal_Ipps_degrees := UDINT_TO_REAL(#read3.nominal_Ipps_degrees) / 1000;
       #out3.nominal_Inps_degrees := UDINT_TO_REAL(#read3.nominal_Inps_degrees) / 1000;
   END_IF;

   #mb_query(data_addr := 40112,
             data_ptr := #read4);
   IF #mb_query.Done THEN
       FOR #c := 1 TO 3 DO
           #out4.active_power[#c] := UDINT_TO_REAL(#read4.active_power[#c]) / 1000;
           #out4.reactive_power[#c] := UDINT_TO_REAL(#read4.reactive_power[#c]) / 1000;
           #out4.apparent_power[#c] := UDINT_TO_REAL(#read4.apparent_power[#c]) / 1000;
           #out4.power_factor[#c] := UDINT_TO_REAL(#read4.power_factor[#c]) / 1000;
       END_FOR;
       #out4.active_power_tot := UDINT_TO_REAL(#read4.active_power_tot) / 1000;
       #out4.reactive_power_tot := UDINT_TO_REAL(#read4.reactive_power_tot) / 1000;
       #out4.apparent_power_tot := UDINT_TO_REAL(#read4.apparent_power_tot) / 1000;
       #out4.power_factor_tot := UDINT_TO_REAL(#read4.power_factor_tot) / 1000;
   END_IF;

   #mb_query(data_addr := 40144,
             data_ptr := #out5);

   #mb_query(data_addr := 40167,
             data_ptr := #read6);
   IF #mb_query.Done THEN
       FOR #c := 1 TO 3 DO
           #out6.secondary_voltage[#c] := UDINT_TO_REAL(#read6.secondary_voltage[#c]) / 1000;
       END_FOR;
       #out6.fault_records := UDINT_TO_REAL(#read6.fault_records) / 1000;
       #out6.event_records := UDINT_TO_REAL(#read6.event_records) / 1000;
       #out6.waveform_records := UDINT_TO_REAL(#read6.waveform_Records) / 1000;
   END_IF;

   "mb_station_block_footer"(sb := #sb,
                             mb_query := #mb_query);
END_FUNCTION_BLOCK

FUNCTION_BLOCK "Siemens_MAG_6000"   // FB54, SCL
{ S7_Optimized_Access := 'TRUE' }
VERSION : 0.1
   VAR_INPUT
      mb_addr : UInt;
   END_VAR
   VAR_IN_OUT
      mb_query : "mb_query";
   END_VAR
   VAR
      sb : "mb_station_block_udt";
      flow : Struct
         velocity : Real;   // mm/s
         flow : Real;
      END_STRUCT;
      totalizer : Array[1..2] of Real;
      serial_number : String[20];
   END_VAR
BEGIN
   // Siemens - SITRANS F M MAG 6000
   //
   // Expansion module: FDK:085U0234

   "mb_station_block_header"(sb := #sb, mb_query := #mb_query);
   #mb_query.mb_addr := #mb_addr;

   #mb_query.mode := #mb_query.c.read.holding_reg;
   #mb_query(data_addr := 3000, data_ptr := #flow);
   #mb_query(data_addr := 3022, data_ptr := #totalizer);
   #mb_query(data_addr := 2520, data_ptr := #serial_number);

   "mb_station_block_footer"(sb := #sb, mb_query := #mb_query);
END_FUNCTION_BLOCK

FUNCTION_BLOCK "Siemens_MASS_6000"   // FB55, SCL
{ S7_Optimized_Access := 'TRUE' }
VERSION : 0.1
   VAR_INPUT
      mb_addr : UInt;
   END_VAR
   VAR_IN_OUT
      mb_query : "mb_query";
   END_VAR
   VAR
      sb : "mb_station_block_udt";
      read : Struct
         value : Real;   // [kg/s or mm/s]
         volumeflow : Real;   // [m3/s]
         density : Real;   // [kg/m3]
         temperature : Real;   // [°C]
         fraction : Array[1..2] of Real;   // [kg/s]
         percent_fraction : Real;   // [%]
         totalizer_1 : Array[1..2] of UDInt;   // [kg or m3]
         totalizer_2 : Array[1..2] of UDInt;   // [kg or m3]
         totalizer_real : Array[1..2] of Real;   // [m3 or kg]
      END_STRUCT;
      serial_number : String[20];
      write1 : Array[1..2] of Struct
         totalizer_selection : UInt;   // 1=Massflow, 2=Fraction A, 3=Fraction B, 4=Volumeflow .
         totalizer_direction : UInt;   // 0=Reverse, 1=Forward, 2=Net
      END_STRUCT;
      write2 : Struct
         low_flow_cut : Real := 0.02;   // (e.g. value 0,02 = 2 %)
         Empty_pipe_limit : Real := 0.0;   // (kg/m3)
         Empty_pipe : Word;   // 0=Off, 1=On
      END_STRUCT;
      write3_noise_filter : UInt := 3;   // 1=min...5=max
      first_scan : Bool := true;
   END_VAR
   // write1[1].totalizer_direction := 1;
   // write1[2].totalizer_direction := 1;
   // write1[1].totalizer_selection := 1;
   // write1[2].totalizer_selection := 4;
   // sb.conf.read_only := true;
BEGIN
   // Siemens 
   // - MASS 6000
   // - MAG 6000
   //
   // Expansion module: FDK:085U0234
   // https://cache.industry.siemens.com/dl/files/906/44880906/att_70364/v1/USMII_MODBUS_AOM_OI_En_en-US.pdf

   IF #first_scan THEN
       #sb.conf.read_only := true;
       #first_scan := false;
   END_IF;

   "mb_station_block_header"(sb := #sb, mb_query := #mb_query);
   #mb_query.mb_addr := #mb_addr;

   #mb_query.mode := #mb_query.c.read.holding_reg;
   #mb_query(data_addr := 3000, data_ptr := #read);
   #mb_query(data_addr := 2520, data_ptr := #serial_number);

   #mb_query.mode := #mb_query.c.write.holding_reg;
   #mb_query(data_addr := 2100, data_ptr := #write1);
   // #mb_query(data_addr := 2025, data_ptr := #write2);
   #mb_query(data_addr := 2030, data_ptr := #write3_noise_filter);

   "mb_station_block_footer"(sb := #sb, mb_query := #mb_query);
END_FUNCTION_BLOCK

FUNCTION_BLOCK "Siemens_sed2_modbus2"   // FB57, SCL
{ S7_Optimized_Access := 'TRUE' }
VERSION : 0.1
   VAR_INPUT
      mb_addr : UInt;
      ref : Real;   // 0-100% ( -100% reverse)
   END_VAR
   VAR_OUTPUT
      speed : Real;   // rpm
      current : Real;   // A x10
      torque : Real;   // Nm x10
      actual_pwr : Real;   // kW x100
      total_kwh : Real;   // kWh
      dc_bus_volt : Real;   // V
   END_VAR
   VAR_IN_OUT
      mb_query : "mb_query";
   END_VAR
   VAR
      sb : "mb_station_block_udt";
      write1 : Struct
         wdog_time : UInt := 1500;   // [ms]
         wdog_action : Word := 1;   // 1:stop, 0:no action
         freq_ref : UInt;
         run_enable : UInt;
         reverse : UInt;
         cmd_start : UInt;
         fault_ack : UInt;
      END_STRUCT;
      write2 : Struct
         current_limit : UInt := 4000;   // A x0
         accel_time : UInt := 1000;   // s x100
         decel_time : UInt := 1000;   // s x100
         manual : UInt;
      END_STRUCT;
      write3 : Struct
         freq_max : UInt := 5000;   // HZ x100
      END_STRUCT;
      read1 : Struct
         freq_output : UInt;   // Hz x10
         speed : UInt;   // rpm
         current : UInt;   // A x10
         torque : UInt;   // Nm x10
         actual_pwr : UInt;   // kW x100
         total_kwh : UInt;   // kWh
         dc_bus_volt : UInt;   // V
         reference : UInt;   // Hz x10
         rated_pwr : UInt;   // kWx100
         output_volts : UInt;
         reverse : UInt;
         run : UInt;
         at_max_freq : UInt;
         ctrl_mode : UInt;   // 1:SERIAL, 0:LOCAL
         enabled : UInt;
         ready_to_run : UInt;
         analog_in_1 : UInt;
         analog_in_2 : UInt;
      END_STRUCT;
      read2 : Struct
         digital_in : Array[1..6] of UInt;
         fault : UInt;
         last_fault : UInt;
         fault_hist : Array[1..4] of UInt;
         warning : UInt;
         last_warning : UInt;
      END_STRUCT;
   END_VAR
   VAR_TEMP
      "real" : Real;
   END_VAR
BEGIN
   // Siemens - SED2-MODBUS2 - Variable Frequency Drive
   // Modbus RTU Interface Module for SED2 
   // 
   // https://www.downloads.siemens.com/download-center/
   // Download.aspx?pos=download&fct=getasset&id1=A6V10073869

   #write1.reverse := BOOL_TO_UINT(#ref < 0);
   #"real" := NORM_X(MIN := 0, VALUE := #ref, MAX := ABS(100));
   #write1.freq_ref := SCALE_X(MIN := 0, VALUE := #"real", MAX := 16#4000);
   #write1.run_enable := BOOL_TO_UINT(#ref <> 0);
   #write1.cmd_start := BOOL_TO_UINT(#ref <> 0);

   "mb_station_block_header"(sb := #sb,
                             mb_query := #mb_query);
   #mb_query.mb_addr := #mb_addr;

   #mb_query.mode := #mb_query.c.mode.write;
   #mb_query(data_addr := 40001,
             data_ptr := #write1);
   #mb_query(data_addr := 40010,
             data_ptr := #write2);
   #mb_query(data_addr := 40016,
             data_ptr := #write3);

   #mb_query.mode := #mb_query.c.mode.read;
   #mb_query(data_addr := 40024,
             data_ptr := #read1);
   #mb_query(data_addr := 40048,
             data_ptr := #read2);

   "mb_station_block_footer"(sb := #sb,
                             mb_query := #mb_query);

   #speed := UINT_TO_REAL(#read1.speed);
   #current := UINT_TO_REAL(#read1.current) / 10;
   #torque := UINT_TO_REAL(#read1.torque) / 10;
   #actual_pwr := UINT_TO_REAL(#read1.actual_pwr) / 100;
   #total_kwh := UINT_TO_REAL(#read1.total_kwh);
   #dc_bus_volt := UINT_TO_REAL(#read1.dc_bus_volt);
END_FUNCTION_BLOCK

FUNCTION_BLOCK "Siemens_Sinamics_G120"   // FB58, SCL
{ S7_Optimized_Access := 'TRUE' }
VERSION : 0.1
   VAR_INPUT
      mb_addr : UInt;
      ref : Real;
   END_VAR
   VAR_IN_OUT
      mb_query : "mb_query";
   END_VAR
   VAR
      sb : "mb_station_block_udt";
      read : Struct
         stw : Struct
            x08_Speed_setpoint : Bool;   // Actual value deviation within tolerance t_off
            x09_Control_requested : Bool;
            x10_f_or_n_comparison_value_reached_exceeded : Bool;
            x11_I_M_or_P_limit_not_reached : Bool;
            x12 : Bool;
            x13_No_motor_overtemperature_alarm : Bool;
            x14_Motor_rotates_forwards : Bool;   // 0 = Motor rotates backwards (n_act < 0)
            x15_No_alarm_thermal_overload_power_unit : Bool;
            x00_Ready_to_power_up : Bool;
            x01_Ready_to_operate : Bool;   // (DC link loaded, pulses blocked)
            x02_Operation_enabled : Bool;   // (drive follows n_set)
            x03_Fault_present : Bool;
            x04_No_coast_down_active : Bool;   // (OFF2 inactive)
            x05_No_fast_stop_active : Bool;   // (OFF3 inactive)
            x06_power_on_inhibit_active : Bool;
            x07_Alarm_present : Bool;
         END_STRUCT;
         actual : Int;
      END_STRUCT;
      write : Struct
         ctw : Struct
            x08 : Bool;
            x09 : Bool;
            x10_control_via_PLC : Bool := TRUE;
            x11_reversal : Bool;
            x12 : Bool;
            x13_Motorized_potentiometer_setpoint_raise : Bool;
            x14_Motorized_potentiometer_setpoint_lower : Bool;
            x15 : Bool;
            x00_R_TRIG_ON : Bool;   // 0 = OFF1 (braking with ramp-function generator, then pulse cancllation &ready-to-power-up)
            x01_No_OFF2 : Bool := TRUE;   // enable is possible. 0 = OFF2 (immediate pulse cancellation and power-on inhibit)
            x02_No_OFF3 : Bool := TRUE;   // enable is possible. 0 = OFF3 braking with the OFF3 ramp p1135, then pulse cancellation andpower-on inhibit)
            x03_Enable_operation : Bool := TRUE;   // (pulses can be enabled) 0 = Inhibit operation (cancel pulses)
            x04_Operating_condition : Bool;   // (the ramp-function generator can be enabled)0 = Inhibit ramp-function generator (set the ramp-function generator output tozero)
            x05_Enable_the_ramp_function_generator : Bool;   // 0 = Stop the ramp-function generator (freeze the ramp-function generatoroutput)
            x06_enable_setpoint : Bool := TRUE;   // 0 = Inhibit setpoint (set the ramp-function generator input to zero)
            x07_R_TRIG_acknowledge_faults : Bool;
         END_STRUCT;
         setpoint : Int;
      END_STRUCT;
   END_VAR
BEGIN
   // Siemens - SINAMICS G120
   // 
   // Web: https://cache.industry.siemens.com/dl/files/944/
   // 35928944/att_7966/v1/application_cu230_modbus_v1_2_en.pdf

   "mb_station_block_header"(sb := #sb, mb_query := #mb_query);
   #mb_query.mb_addr := #mb_addr;

   #mb_query.mode := #mb_query.c.read.holding_reg;
   #mb_query(data_addr := 40110, data_ptr := #read);

   #write.ctw.x00_R_TRIG_ON :=
   (* *)#ref <> 0
   (* *)AND NOT #read.stw.x07_Alarm_present
   (* *)AND #read.stw.x01_Ready_to_operate
   (* *)AND #read.stw.x00_Ready_to_power_up;
   #write.setpoint := REAL_TO_INT(#ref);

   #mb_query.mode := #mb_query.c.write.holding_reg;
   #mb_query(data_addr := 40100, data_ptr := #write);

   "mb_station_block_footer"(sb := #sb, mb_query := #mb_query);
END_FUNCTION_BLOCK

FUNCTION_BLOCK "Siemens_SITRANS_F_M_MAG_8000"   // FB59, SCL
{ S7_Optimized_Access := 'TRUE' }
VERSION : 0.1
   VAR_INPUT
      mb_addr : UInt;
   END_VAR
   VAR_IN_OUT
      mb_query : "mb_query";
   END_VAR
   VAR
      sb : "mb_station_block_udt";
      flow : Struct
         velocity : Real;   // mm/s
         flow : Real;
      END_STRUCT;
      totalizer : Array[1..3] of UDInt;
   END_VAR
BEGIN
   // Siemens - SITRANS F M MAG 8000
   // https://cache.industry.siemens.com/dl/files/509/54091509/
   // att_100244/v1/A5E03409989_01_MAG8000_MODBUS_AOM_OI_.pdf

   "mb_station_block_header"(sb := #sb, mb_query := #mb_query);
   #mb_query.mb_addr := #mb_addr;

   #mb_query.mode := #mb_query.c.read.holding_reg;
   #mb_query(data_addr := 2999, data_ptr := #flow);
   #mb_query(data_addr := 3016, data_ptr := #totalizer);

   "mb_station_block_footer"(sb := #sb, mb_query := #mb_query);
END_FUNCTION_BLOCK

FUNCTION_BLOCK "Siemens_vav_compact_controller"   // FB60, SCL
{ S7_Optimized_Access := 'TRUE' }
VERSION : 0.1
   VAR_INPUT
      mb_addr : UInt;
      sp : Real;   // setpoint
      sp_backup : Real;
   END_VAR
   VAR_IN_OUT
      mb_query : "mb_query";
   END_VAR
   VAR
      sb : "mb_station_block_udt";
      read : Struct
         Actual_position : Int;
         Actual_Flow_rel : UInt;
         Actual_Flow_abs : UInt;
         Actual_Pressure : UInt;
      END_STRUCT;
      write1 : Struct
         Setpoint : Int;
      END_STRUCT;
      write2 : Struct
         backup_mode : Int := 0;
         backup_position : Int := 0;
      END_STRUCT;
   END_VAR
BEGIN
   // Siemens - VAV compact controller 
   // GDB181.1E/MO Operating voltage AC 24 V, 5 Nm
   // GLB181.1E/MO Operating voltage AC 24 V, 10 Nm

   // https://www.micromatic.no/globalassets/inriver/resources/
   // bruksanvisning_ko1320-28.pdf

   "mb_station_block_header"(sb := #sb, mb_query := #mb_query);
   #mb_query.mb_addr := #mb_addr;

   #mb_query.mode := #mb_query.c.read.holding_reg;
   #mb_query(data_addr := 3, data_ptr := #read);

   #mb_query.mode := #mb_query.c.write.holding_reg;
   #write1.Setpoint := REAL_TO_INT(#sp) * 100;
   #mb_query(data_addr := 1, data_ptr := #write1);
   #write2.backup_position := REAL_TO_INT(#sp_backup) * 100;
   #mb_query(data_addr := 513, data_ptr := #write2);

   "mb_station_block_footer"(sb := #sb, mb_query := #mb_query);

   (*
   Backup mode (write 2)
   0 = Go to BackupPosition
   1 = Keep last position
   2 = Disabled
   *)
END_FUNCTION_BLOCK

FUNCTION_BLOCK "Siemens_SIWAREX_WP251"   // FB93, SCL
{ S7_Optimized_Access := 'TRUE' }
VERSION : 0.1
   VAR_INPUT
      mb_addr : UInt;
   END_VAR
   VAR_IN_OUT
      mb_query : "mb_query";
   END_VAR
   VAR
      sb : "mb_station_block_udt";
      read1 : Struct
         Unit_of_weight : UInt;   // x1000
         Gross_identifier : UInt;
         Code_for_regulations : UInt;
         Reserve : UInt;
         weighing_range_min : UInt;
         weighing_range_max : Real;
         Calibration_weight : Array[0..2] of Real;
         Calibration_digits : Array[0..2] of Real;
         Scale_interval : Array[0..2] of Real;   // (Page 64)
      END_STRUCT;
      read2 : Struct
         stat : Struct
            x08 : Bool;
            x09 : Bool;
            x10 : Bool;
            x11 : Bool;
            x12 : Bool;
            x13 : Bool;
            x14 : Bool;
            x15 : Bool;
            x00 : Bool;
            x01 : Bool;
            x02 : Bool;
            x03 : Bool;
            x04 : Bool;
            x05 : Bool;
            x06 : Bool;
            x07 : Bool;
         END_STRUCT;
         Reserve : UInt;
         Max_tare_load : Real;
         Max_negative_zero_limit_power_on : Real;
         Max_positive_zero_limit_power_on : Real;
         Max_negative_zero_limit_semi_automatically : Real;
         Max_positive_zero_limit_semi_automatically : Real;
      END_STRUCT;
      read3 : Struct
         standstill : Array[1..2] of Struct
            range : Real;
            "time" : Time;
            max_waiting_time : Time;
         END_STRUCT;
         frequency_low_pass_filter1 : Real;
         Order_no_low_pass_filter1 : UInt;
         depth_average_filter : UInt;
         reserve_1 : UInt;
         weighing_operating_mode : UInt;
         resolution_of_master_totalizer : Real;
         Reserve_2 : Real;
         SecureDisplay_including_weighing_range_data : UInt;
      END_STRUCT;
      read4 : Struct
         SecureDisplay_interface : UInt;   // (Page 71)
         String_header_version_SecureDisplay : String[2];
         SecureDisplay_version : String[12];
         Minimum_zoom_factor_of_SecureDisplay : UInt;
         Reserve_1 : Array[1..3] of Real;
         Reserve_2 : Array[1..3] of UInt;
         Grid_frequency : UInt;   // 0: 50 Hz, 1: 60Hz
      END_STRUCT;
      write1 : Struct
         Smallest_weight_below_TU2 : Real;
         Highest_weight_above_TH2 : Real;
         Single_setpoin : Real;
         Net_weight_average_value : Real;
         Standard_deviation : Real;
      END_STRUCT;
   END_VAR
BEGIN
   // Siemens - SIWAREX WP251 - Electronic Weighing System
   // A5E37203357A
   // 
   // https://cache.industry.siemens.com/dl/files/751/109481751/att_893477/v1/Manual_SIWAREX_WP251_en_en-US.pdf

   "mb_station_block_header"(sb := #sb, mb_query := #mb_query);
   #mb_query.mb_addr := #mb_addr;

   #mb_query.mode := #mb_query.c.read.holding_reg;
   #mb_query(data_addr := 1011, data_ptr := #read1);
   #mb_query(data_addr := 1032, data_ptr := #read2);
   #mb_query(data_addr := 1044, data_ptr := #read3);
   #mb_query(data_addr := 1067, data_ptr := #read4);

   #mb_query.mode := #mb_query.c.write.holding_reg;
   #mb_query(data_addr := 4101, data_ptr := #write1);

   "mb_station_block_footer"(sb := #sb, mb_query := #mb_query);

   (*
   Unit of weight:
   0: "mg"
   1: "g"
   2: "kg"
   3: "t"
   4: "oz" (ounce)
   5: "lb" (pound)
   6: "T" (=short tons)
   7: "TL" (= long tons)

   Gross identifier:
   0: "brutto" 
   1: "Gross"

   Code for regulations:
   0: None
   1: OIML

   Weighing operating mode (Page 71):
   0: NAWI – Filling
   1: NAWI – Removal
   10: AWI
   20: ACI – Filling 
   21: ACI – Removal

   *)
END_FUNCTION_BLOCK

// folder: Library/Modbus/Station blocks/sb Untested/S/Swan

FUNCTION_BLOCK "Swan_AMI_CACE"   // FB65, SCL
{ S7_Optimized_Access := 'TRUE' }
VERSION : 0.1
   VAR_INPUT
      mb_addr : USInt;
   END_VAR
   VAR_IN_OUT
      mb_query : "mb_query";
   END_VAR
   VAR
      sb : "mb_station_block_udt";
      data : Struct
         cond_sc : Array[1..3] of Real;   // µS
         Temp : Array[1..3] of Real;
         flow : Real;
         pH : Real;
         alkalyzer : Real;
         cond_uc : Array[1..3] of Real;
         Pt1000_Temp : Array[1..3] of Real;
         raw_flow : Real;
         case_temperature : Real;
         EDI_voltage : Real;
         EDI_current : Real;
         Degasser_temperature : Real;
         Degasser_boiling_point : Real;
         Degasser_PWM : Real;
         Degasser_line_voltage : Real;
         Degasser_air_pressure : Real;
         Degasser_Case_Temp : Real;
         signal_output : Array[1..2] of Real;
         "Instrument Display Status" : DWord;
      END_STRUCT;
      alarm : Struct
         x00_Cond_1_Alarm_high : Bool;
         x01_Cond_1_Alarm_low : Bool;
         x02_Cond_2_Alarm_high : Bool;
         x03_Cond_2_Alarm_low : Bool;
         x04_Cond_3_Alarm_high : Bool;
         x05_Cond_3_Alarm_low : Bool;
         x06_Temp_1_high : Bool;
         x07_Temp_1_low : Bool;
         x08_sample_flow_high : Bool;
         x09_sample_flow_low : Bool;
         x10_temp_1_shorted : Bool;
         x11_temp_1_disconnected : Bool;
         x12_case_temp_high : Bool;
         x13_case_temp_low : Bool;
         x14_pH_Error : Bool;
         x15_Degasser_frontend : Bool;
         x16_control_timeout : Bool;
         x17_Degasser_disconnected : Bool;
         x18_Temp_2_shorted : Bool;
         x19_Temp_2_disconnected : Bool;
         x20_Temp_3_shorted : Bool;
         x21_Temp_3_disconnected : Bool;
         x22_Degasser_Ctl_Timeout : Bool;
         x23_Input_Active : Bool;
         x24_IC_MK41T56 : Bool;
         x25_IC_LM75 : Bool;
         x26_IC_PCF8574 : Bool;
         x27_Signal_output_open : Bool;
         x28_Calibration_Degasser : Bool;
         x29_EEprom_Front_end : Bool;
         x30_Calibration_Recout : Bool;
         x31_Wrong_Front_end : Bool;
         x32_pH_Alarm_high : Bool;
         x33_pH_Alarm_low : Bool;
         x34_Alkali_Alarm_high : Bool;
         x35_Alkali_Alarm_low : Bool;
         x36_Temp_2_high : Bool;
         x37_Temp_2_low : Bool;
         x38_Temp_3_high : Bool;
         x39_Temp_3_low : Bool;
         x40_Degasser_Line_Voltage : Bool;
         x41_Degasser_Temperature : Bool;
         x42_EDI_out_of_range : Bool;
         x43_No_sample_flow : Bool;
         x44_EDI_DAC_disconnected : Bool;
         "x45_ EDI_ADC_disconnected" : Bool;
         x46 : Bool;
         x47_EDI_module_exhausted : Bool;
      END_STRUCT;
      write : Struct
         x0_relay_contacts_1 : Bool;
         x1_relay_contacts_2 : Bool;
         x2 : Bool;
         x3 : Bool;
         x4 : Bool;
         x5 : Bool;
         x6 : Bool;
         x7 : Bool;
      END_STRUCT;
   END_VAR
BEGIN
   // Swan - AMI CACE - Conductivity measurement 
   // Swan analytical instruments
   // http://www.swan.ch/GetAttachment.axd?attaName=e82f8e94-ab32-4930-8c9d-a56dc0847f61
   // Page 9

   "mb_station_block_header"(sb := #sb,
                             mb_query := #mb_query);
   #mb_query.mb_addr := #mb_addr;
   #mb_query.data_addr := 0;

   #mb_query(mode := #mb_query.c.read.input_reg,
             data_ptr := #data);

   #mb_query(mode := #mb_query.c.read.discrete_input,
             data_ptr := #alarm);

   (*#mb_query(mode := #mb_query.c.write.discrete_output,
             data_len := 2,
             data_ptr := #write);*)

   "mb_station_block_footer"(sb := #sb,
                             mb_query := #mb_query);
END_FUNCTION_BLOCK

FUNCTION_BLOCK "Swan_AMI_Codes-II_CC"   // FB66, SCL
{ S7_Optimized_Access := 'TRUE' }
VERSION : 0.1
   VAR_INPUT
      mb_addr : USInt;
   END_VAR
   VAR_IN_OUT
      mb_query : "mb_query";
   END_VAR
   VAR
      sb : "mb_station_block_udt";
      data : Struct
         free_available_chlorine : Real;   // ppm
         total_chlorine_1_tc1 : Real;   // ppm
         total_chlorine_2_tc2 : Real;   // ppm
         calculated_monochloramine : Real;   // ppm
         calculated_combined_chlorine : Real;   // ppm
         calculated_dichloramine : Real;   // ppm
         temperature : Real;   // °C
         flow : Real;   // B/s
         pH : Real;   // pH
         absorbance : Real;
         photometer_frequency : Real;   // Hz
         remaining_DPD_buffer : Real;   // %
         remaining_potassium_Iodide : Real;   // %
         remaining_cleaning_solution : Real;   // %
         raw_temp_NTK5 : Real;   // Ohm
         raw_flow : Real;   // Hz
         raw_pH : Real;   // mV
         case_temperature : Real;   // °C
         signal_output_1 : Real;   // mA
         signal_output_2 : Real;   // mA
         instrument_display_status : Real;
      END_STRUCT;
      alarm : Struct
         x00_high_fac : Bool;
         x01_low_fac : Bool;
         x02_high_tc1 : Bool;
         x03_low_tc1 : Bool;
         x04_high_tc2 : Bool;
         x05_low_tc2 : Bool;
         x06_sample_temp_high : Bool;
         x07_sample_temp_low : Bool;
         x08_sample_flow_high : Bool;
         x09_sample_flow_low : Bool;
         x10_Temp_shorted : Bool;
         x11_Temp_disconnected : Bool;
         x12_case_temp_high : Bool;
         x13_case_temp_low : Bool;
         x14_valve_1_defective : Bool;
         x15_dis_invalid : Bool;
         x16_control_timeout : Bool;
         x17_reagent_pump : Bool;
         x18_photometer_not_connected : Bool;
         x19_photometer_dirty : Bool;
         x20_absorbance_too_high : Bool;
         x21_reagent_empty : Bool;
         x22_cleaning_reagent : Bool;
         x23_input_active : Bool;
         x24_IC_MK41T56 : Bool;
         x25_IC_LM75 : Bool;
         x26_IC_PCF8574 : Bool;
         x27_signal_output_open : Bool;
         x28_EEprom_motherboard : Bool;
         x29_EEprom_front_end : Bool;
         x30_calibration_recout : Bool;
         x31_wrong_front_end : Bool;
         x32_high_cmc : Bool;
         x33_low_cmc : Bool;
         x34_high_ccc : Bool;
         x35_low_ccc : Bool;
         x36_high_cdc : Bool;
         x37_low_cdc : Bool;
         x38_high_pH : Bool;
         x39_low_pH : Bool;
         x40_DPD_buffer : Bool;
         x41_potassium_Iodide : Bool;
         x42_cleaning_solution : Bool;
         x43 : Bool;
         x44 : Bool;
         x45 : Bool;
         x46 : Bool;
         x47 : Bool;
      END_STRUCT;
      write : Struct
         x0_relay_contacts_1 : Bool;
         x1_relay_contacts_2 : Bool;
         x2_hold : Bool;
         x3_Remote_off : Bool;
         x4 : Bool;
         x5 : Bool;
         x6 : Bool;
         x7 : Bool;
      END_STRUCT;
   END_VAR
BEGIN
   // Swan - AMI Codes-II CC
   //
   // http://www.swan.ch/GetAttachment.axd?attaName=e82f8e94-ab32-4930-8c9d-a56dc0847f61
   // Page 17

   "mb_station_block_header"(sb := #sb,
                             mb_query := #mb_query);
   #mb_query.mb_addr := #mb_addr;
   #mb_query.data_addr := 0;

   #mb_query(mode := #mb_query.c.read.input_reg,
             data_ptr := #data);

   #mb_query(mode := #mb_query.c.read.discrete_input,
             data_ptr := #alarm);

   (*#mb_query(mode := #mb_query.c.write.discrete_output,
             data_len := 4,
             data_ptr := #write);*)

   "mb_station_block_footer"(sb := #sb,
                             mb_query := #mb_query);
END_FUNCTION_BLOCK

FUNCTION_BLOCK "Swan_AMI_Hydrogen"   // FB67, SCL
{ S7_Optimized_Access := 'TRUE' }
VERSION : 0.1
   VAR_INPUT
      mb_addr : USInt;
   END_VAR
   VAR_IN_OUT
      mb_query : "mb_query";
   END_VAR
   VAR
      sb : "mb_station_block_udt";
      data : Struct
         hydrogen : Real;   // ppb
         temperature : Real;   // °C
         flow : Real;   // l/h
         saturation : Real;   // %
         air_pressure : Real;   // hPa
         raw_Current_temp_compensated : Real;   // nA
         raw_current_uncompensated : Real;   // nA
         raw_temp_Pt1000 : Real;   // Ω
         raw_flow : Real;   // Hz
         reserved : Real;
         case_temperature : Real;   // °C
         signal_output_1 : Real;   // mA
         signal_output_2 : Real;   // mA
         instrument_display_status : UDInt;
      END_STRUCT;
      alarm : Struct
         x00_hydrogen_alarm_high : Bool;
         x01_hydrogen_alarm_low : Bool;
         x02_saturation_alarm_high : Bool;
         x03_saturation_alarm_low : Bool;
         x04 : Bool;
         x05 : Bool;
         x06_sample_temp_high : Bool;
         x07_sample_temp_low : Bool;
         x08_sample_flow_high : Bool;
         x09_sample_flow_low : Bool;
         x10_temp_shorted : Bool;
         x11_temp_disconnected : Bool;
         x12_case_temp_high : Bool;
         x13_case_temp_low : Bool;
         x14 : Bool;
         x15 : Bool;
         x16_control_timeout : Bool;
         x17_faraday_efficiency_QED : Bool;
         x18_quality_assurance : Bool;
         x19 : Bool;
         x20 : Bool;
         x21 : Bool;
         x22 : Bool;
         x23_input_active : Bool;
         x24_IC_MK41T56 : Bool;
         x25_IC_LM75 : Bool;
         x26_IC_PCF8574 : Bool;
         x27_Signal_output_open : Bool;
         x28_EEprom_Motherboard : Bool;
         x29_EEprom_Front_end : Bool;
         x30_Calibration_Recout : Bool;
         x31_Wrong_Front_end : Bool;
         x32 : Bool;
         x33 : Bool;
         x34 : Bool;
         x35 : Bool;
         x36 : Bool;
         x37 : Bool;
         x38 : Bool;
         x39 : Bool;
         x40 : Bool;
         x41 : Bool;
         x42 : Bool;
         x43 : Bool;
         x44 : Bool;
         x45 : Bool;
         x46 : Bool;
         x47_Status_Electrolyte_depleted : Bool;
      END_STRUCT;
      write : Struct
         x0_relay_contacts_1 : Bool;
         x1_relay_contacts_2 : Bool;
         x2_hold : Bool;
         x3_Remote_off : Bool;
         x4 : Bool;
         x5 : Bool;
         x6 : Bool;
         x7 : Bool;
      END_STRUCT;
   END_VAR
BEGIN
   // Swan - AMI Hydrogen
   // Swan analytical instruments
   // http://www.swan.ch/GetAttachment.axd?attaName=e82f8e94-ab32-4930-8c9d-a56dc0847f61
   // Page 37

   "mb_station_block_header"(sb := #sb,
                             mb_query := #mb_query);
   #mb_query.mb_addr := #mb_addr;
   #mb_query.data_addr := 0;

   #mb_query(mode := #mb_query.c.read.input_reg,
             data_ptr := #data);

   #mb_query(mode := #mb_query.c.read.discrete_input,
             data_ptr := #alarm);

   (*#mb_query(mode := #mb_query.c.write.discrete_output,
             data_len := 4,
             data_ptr := #write);*)

   "mb_station_block_footer"(sb := #sb,
                             mb_query := #mb_query);
END_FUNCTION_BLOCK

FUNCTION_BLOCK "Swan_AMI_Oxysafe"   // FB68, SCL
{ S7_Optimized_Access := 'TRUE' }
VERSION : 0.1
   VAR_INPUT
      mb_addr : USInt;
   END_VAR
   VAR_IN_OUT
      mb_query : "mb_query";
   END_VAR
   VAR
      sb : "mb_station_block_udt";
      data : Struct
         oxygen : Real;   // ppm
         temperature : Real;   // °C
         flow : Real;   // l/h
         saturation : Real;   // %
         air_pressure : Real;   // hPa
         raw_Oxygen_temp_compensated : Real;   // nA
         raw_oxygen_temp_uncompensated : Real;   // nA
         raw_Temp_Pt1000 : Real;   // Ohm
         raw_flow : Real;   // Hz
         remaining_electrolyte : Real;   // %
         case_temperature : Real;   // °C
         signal_output_1 : Real;   // mA
         signal_output_2 : Real;   // mA
         instrument_display_status : DWord;
      END_STRUCT;
      alarm : Struct
         x00_Oxygen_alarm_high : Bool;
         x01_Oxygen_alarm_low : Bool;
         x02_Saturation_alarm_high : Bool;
         x03_Saturation_alarm_low : Bool;
         x04 : Bool;
         x05 : Bool;
         x06_Sample_temp_high : Bool;
         x07_Sample_temp_low : Bool;
         x08_sample_flow_high : Bool;
         x09_sample_flow_low : Bool;
         x10_temp_shorted : Bool;
         x11_temp_disconnected : Bool;
         x12_case_temp_high : Bool;
         x13_case_temp_low : Bool;
         x14 : Bool;
         x15 : Bool;
         x16_control_timeout : Bool;
         x17_Faraday_efficiency_QED : Bool;
         x18 : Bool;
         x19 : Bool;
         x20 : Bool;
         x21 : Bool;
         x22 : Bool;
         x23_input_active : Bool;
         x24_IC_MK41T56 : Bool;
         x25_IC_LM75 : Bool;
         x26_IC_PCF8574 : Bool;
         x27_Signal_output_open : Bool;
         x28_EEprom_Motherboard : Bool;
         x29_EEprom_Front_end : Bool;
         x30_Calibration_Recout : Bool;
         x31_Wrong_Front_end : Bool;
         x32 : Bool;
         x33 : Bool;
         x34 : Bool;
         x35 : Bool;
         x36 : Bool;
         x37 : Bool;
         x38 : Bool;
         x39 : Bool;
         x40_Electrolyte_depleted : Bool;
         x41 : Bool;
         x42 : Bool;
         x43 : Bool;
         x44 : Bool;
         x45 : Bool;
         x46 : Bool;
         x47 : Bool;
      END_STRUCT;
      write : Struct
         x0_relay_contacts_1 : Bool;
         x1_relay_contacts_2 : Bool;
         x2_hold : Bool;
         x3_Remote_off : Bool;
         x4 : Bool;
         x5 : Bool;
         x6 : Bool;
         x7 : Bool;
      END_STRUCT;
   END_VAR
BEGIN
   // Swan - AMI - Oxysafe
   // Swan analytical instruments
   // http://www.swan.ch/GetAttachment.axd?attaName=e82f8e94-ab32-4930-8c9d-a56dc0847f61
   // Page 53

   "mb_station_block_header"(sb := #sb,
                             mb_query := #mb_query);
   #mb_query.mb_addr := #mb_addr;
   #mb_query.data_addr := 0;

   #mb_query(mode := #mb_query.c.read.input_reg,
             data_ptr := #data);

   #mb_query(mode := #mb_query.c.read.discrete_input,
             data_ptr := #alarm);

   (*#mb_query(mode := #mb_query.c.write.discrete_output,
             data_len := 4,
             data_ptr := #write);*) 

   "mb_station_block_footer"(sb := #sb,
                             mb_query := #mb_query);
END_FUNCTION_BLOCK

FUNCTION_BLOCK "Swan_AMI_pH-Redox"   // FB69, SCL
{ S7_Optimized_Access := 'TRUE' }
VERSION : 0.1
   VAR_INPUT
      mb_addr : USInt;
   END_VAR
   VAR_IN_OUT
      mb_query : "mb_query";
   END_VAR
   VAR
      sb : "mb_station_block_udt";
      data : Struct
         pH_Redox : Real;   // pH/mV
         temperature : Real;   // °C
         Flow : Real;   // l/h
         raw_signal : Real;   // mV
         Pt_1000_temp : Real;   // ohm
         raw_flow : Real;   // Hz
         sensor_check : Real;   // Mohm
         case_temperature : Real;   // °C
         signal_output_1 : Real;   // mA
         signal_output_2 : Real;   // mA
         instrument_display_status : DWord;
      END_STRUCT;
      alarm : Struct
         x00_alarm_high : Bool;
         x01_alarm_low : Bool;
         x02 : Bool;
         x03 : Bool;
         x04 : Bool;
         x05 : Bool;
         x06_sample_temp_high : Bool;
         x07_sample_temp_low : Bool;
         x08_sample_flow_high : Bool;
         x09_sample_flow_low : Bool;
         x10_temp_shorted : Bool;
         x11_temp_disconnected : Bool;
         x12_case_temp_high : Bool;
         x13_case_temp_low : Bool;
         x14 : Bool;
         x15 : Bool;
         x16_control_timeout : Bool;
         x17 : Bool;
         x18 : Bool;
         x19 : Bool;
         x20 : Bool;
         x21 : Bool;
         x22 : Bool;
         x23_input_active : Bool;
         x24_IC_MK41T56 : Bool;
         x25_IC_LM75 : Bool;
         x26_IC_PCF8574 : Bool;
         x27_Signal_output_open : Bool;
         x28_EEprom_Motherboard : Bool;
         x29_EEprom_Front_end : Bool;
         x30_Calibration_Recout : Bool;
         x31_Wrong_Front_end : Bool;
      END_STRUCT;
      write : Struct
         x0_relay_contacts_1 : Bool;
         x1_relay_contacts_2 : Bool;
         x2_hold : Bool;
         x3_Remote_off : Bool;
         x4 : Bool;
         x5 : Bool;
         x6 : Bool;
         x7 : Bool;
      END_STRUCT;
   END_VAR
BEGIN
   // Swan - AMI pH-Redox
   // Swan analytical instruments
   // 
   // http://www.swan.ch/GetAttachment.axd?attaName=e82f8e94-ab32-4930-8c9d-a56dc0847f61
   // Page 73

   "mb_station_block_header"(sb := #sb, mb_query := #mb_query);
   #mb_query.mb_addr := #mb_addr;
   #mb_query.data_addr := 0;

   #mb_query(mode := #mb_query.c.read.input_reg,
             data_ptr := #data);

   #mb_query(mode := #mb_query.c.read.discrete_input,
             data_ptr := #alarm);

   (*#mb_query(mode := #mb_query.c.write.discrete_output,
             data_len := 4,
             data_ptr := #write);*)

   "mb_station_block_footer"(sb := #sb, mb_query := #mb_query);
END_FUNCTION_BLOCK

// folder: Library/Modbus/Station blocks/sb Untested/V

FUNCTION_BLOCK "Vacon_OPTC2_C8"   // FB72, SCL
{ S7_Optimized_Access := 'TRUE' }
VERSION : 0.1
   VAR_INPUT
      mb_addr : UInt;
      ref : Real;
   END_VAR
   VAR_OUTPUT
      actual_speed : Real;
      Output_Frequency : Real;   // hz
      Motor_Speed : Real;   // rpm
      Motor_Current : Real;   // A
      Motor_Torque : Real;   // %
      Motor_Power : Real;   // %
      Motor_Voltage : Real;   // V
      DC_link_voltage : Real;   // V
   END_VAR
   VAR_IN_OUT
      mb_query : "mb_query";
   END_VAR
   VAR
      sb : "mb_station_block_udt";
      write : Struct
         ctw : Struct
            byte0 : Bool;
            x00_run : Bool;
            x01_reverse : Bool;
            x02_reset : Bool;
            x03 : Bool;
            x04 : Bool;
            x05 : Bool;
            x06 : Bool;
            x07 : Bool;
         END_STRUCT;
         "General Control Word" : Word;
         speed_reference : Int;
      END_STRUCT;
      read : Struct
         status : Struct
            tc_speed_limit_not_active : Bool;   // [08]
            detected_encoder_direction_counterclockwise : Bool;   // [09]
            UV_fast_stop_not_active : Bool;   // [10]
            x11 : Bool;   // [11]
            x12 : Bool;   // [12]
            x13 : Bool;   // [13]
            x14 : Bool;   // [14]
            x15 : Bool;   // [15]
            ready : Bool;   // [00]
            RUN : Bool;   // [01]
            reverse : Bool;   // [02]
            faulted : Bool;   // [03]
            warning : Bool;   // [04]
            ref_frequency_reached : Bool;   // [05]
            motor_is_running_at_zero_speed : Bool;   // [06]
            flux_ready : Bool;   // [07]
         END_STRUCT;
         general_status : Struct
            x08 : Bool;
            x09 : Bool;
            x10 : Bool;
            x11 : Bool;
            x12 : Bool;
            x13_Fieldbus_control : Bool;
            "x14_Panel control" : Bool;
            x15_IO_control : Bool;
            x00 : Bool;
            x01 : Bool;
            x02 : Bool;
            x03 : Bool;
            x04 : Bool;
            x05 : Bool;
            x06 : Bool;
            x07 : Bool;
         END_STRUCT;
         actual_speed : Int;
         Output_Frequency : Int;   // 0.01 Hz
         Motor_Speed : Int;   // 1 rpm
         Motor_Current : Int;   // 0.1 A
         Motor_Torque : Int;   // 0.1 %
         Motor_Power : Int;   // 0.1 %
         Motor_Voltage : Int;   // 0.1 V
         DC_link_voltage : Int;   // 1 V
         Active_Fault_Code : Int;
      END_STRUCT;
   END_VAR
BEGIN
   // Vacon NX - OPTC2/C8 - AC drives
   // Modbus/N2 option board
   // Document code: DPD00899A , Date 19.01.2012
   // Web: http://www.vacon.com/ImageVaultFiles/id_3118/cf_2/
   //      Vacon-NX-OPTC2-C8-Modbus-N2-Board-User-Manual-DPD0.
   //      PDF?635223804391930000

   "mb_station_block_header"(sb := #sb, mb_query := #mb_query);
   #mb_query.mb_addr := #mb_addr;

   #mb_query.mode := #mb_query.c.read.holding_reg;

   #mb_query(data_addr := 42101, data_ptr := #read);
   IF #mb_query.Done THEN
       #actual_speed := INT_TO_REAL(#read.actual_speed);
       #Output_Frequency := INT_TO_REAL(#read.Output_Frequency) * 0.01;
       #Motor_Speed := INT_TO_REAL(#read.Motor_Speed);
       #Motor_Current := INT_TO_REAL(#read.Motor_Current) * 0.1;
       #Motor_Torque := INT_TO_REAL(#read.Motor_Torque) * 0.1;
       #Motor_Power := INT_TO_REAL(#read.Motor_Power) * 0.1;
       #Motor_Voltage := INT_TO_REAL(#read.Motor_Voltage) * 0.1;
       #DC_link_voltage := INT_TO_REAL(#read.DC_link_voltage);
   END_IF;
   // -------------------------------------------------------
   #mb_query.mode := #mb_query.c.write.holding_reg;

   #write.ctw.x00_run := #ref <> 0;
   #mb_query(data_addr := 42001, data_ptr := #write.ctw);
   #write.speed_reference := REAL_TO_INT(#ref * 100);
   #mb_query(data_addr := 42003, data_ptr := #write.speed_reference);

   "mb_station_block_footer"(sb := #sb, mb_query := #mb_query);
END_FUNCTION_BLOCK

FUNCTION_BLOCK "vega_vegabar_81"   // FB73, SCL
{ S7_Optimized_Access := 'TRUE' }
VERSION : 0.1
   VAR_INPUT
      mb_addr : UInt;
   END_VAR
   VAR_IN_OUT
      mb_query : "mb_query";
   END_VAR
   VAR
      sb : "mb_station_block_udt";
      read1 : Struct
         status : Struct
            x08 : Bool;
            x09 : Bool;
            x10 : Bool;
            x11 : Bool;
            x12 : Bool;
            x13 : Bool;
            x14 : Bool;
            x15 : Bool;
            x00_invalid_measurement_1 : Bool;
            x01_invalid_measurement_2 : Bool;
            x02_invalid_measurement_3 : Bool;
            x03_invalid_measurement_4 : Bool;
            x04 : Bool;
            x05 : Bool;
            x06 : Bool;
            x07 : Bool;
         END_STRUCT;
         z : Word;
         data : Array[1..4] of Real;
      END_STRUCT;
   END_VAR
BEGIN
   // Vega - VEGABAR 81

   "mb_station_block_header"(sb := #sb, mb_query := #mb_query);
   #mb_query.mb_addr := #mb_addr;

   #mb_query(mode := #mb_query.c.read.holding_reg,
             data_addr := 2000,
             data_ptr := #read1);

   "mb_station_block_footer"(sb := #sb, mb_query := #mb_query);

   (*
   Unit Code Measurement Unit:
   32 Degree Celsius
   33 Degree Fahrenheit
   40 US Gallon
   41 Liters
   42 Imperial Gallons
   43 Cubic Meters
   44 Feet
   45 Meters
   46 Barrels
   47 Inches
   48 Centimeters
   49 Millimeters
   111 Cubic Yards
   112 Cubic Feet
   113 Cubic Inches
   *)
END_FUNCTION_BLOCK

// folder: Library/Modbus/Station blocks/sb Untested/W

FUNCTION_BLOCK "Weg_CFW100"   // FB74, SCL
{ S7_Optimized_Access := 'TRUE' }
VERSION : 0.1
   VAR_INPUT
      mb_addr : UInt;
   END_VAR
   VAR_IN_OUT
      mb_query : "mb_query";
   END_VAR
   VAR
      sb : "mb_station_block_udt";
      read1 : Struct
         Output_Speed : UInt;   // 2
         Motor_Current : UInt;
         DC_Link_Voltage : UInt;
         Output_Frequency : UInt;
         Inverter_Status : UInt;
         Output_Voltage : UInt;
         Motor_Torque : UInt;
         Active_Current : UInt;
         digital_input : UInt;
      END_STRUCT;
      read2_staus : Struct
         running : Bool;   // [08]
         ready : Bool;   // [09]
         forward : Bool;   // [10]
         jog_active : Bool;   // [11]
         remote_mode : Bool;   // [12]
         undervoltage : Bool;   // [13]
         x14 : Bool;   // [14]
         fault : Bool;   // [15]
         x00 : Bool;   // [00]
         x01 : Bool;   // [01]
         x02 : Bool;   // [02]
         x03 : Bool;   // [03]
         x04 : Bool;   // [04]
         "2nd_Ramp" : Bool;   // 0: 1st Acceleration and deceleration ramp by P100 and P101.
         configuration_state : Bool;   // [06]
         alarm : Bool;   // [07]
         "a" : Struct
            x08 : Bool;
            x09 : Bool;
            x10 : Bool;
            x11 : Bool;
            x12 : Bool;
            x13 : Bool;
            x14 : Bool;
            x15 : Bool;
            x00 : Bool;
            x01 : Bool;
            x02 : Bool;
            x03 : Bool;
            x04 : Bool;
            x05 : Bool;
            x06 : Bool;
            x07 : Bool;
         END_STRUCT;
      END_STRUCT;
      write1 : Struct
         Minimum_Frequency : UInt;
         Maximum_Frequency : UInt := 50;
         Maximum_Output_Current : UInt := 100;
      END_STRUCT;
      write2 : Struct
         "Acceleration Time" : UInt := 5;
         "Deceleration Time" : UInt := 10;
      END_STRUCT;
      write3_sel_rem : UInt := 1;   // 1 = Always Remote
      write4_Ref_sel : UInt := 9;   // 9=serial
      write5 : Struct
         controll_word : Struct
            x08 : Bool;
            x09 : Bool;
            x10 : Bool;
            x11 : Bool;
            x12 : Bool;
            x13 : Bool;
            x14 : Bool;
            x15 : Bool;
            x00_no_ramp_stop : Bool := TRUE;
            x01_start : Bool := TRUE;
            x02_Forward : Bool;
            x03_jog : Bool;
            x04_Remote : Bool := TRUE;
            "x05_2nd Ramp" : Bool;
            x06 : Bool;
            x07_Fault_Reset : Bool;
            "a" : Struct
               x08 : Bool;
               x09 : Bool;
               x10 : Bool;
               x11 : Bool;
               x12 : Bool;
               x13 : Bool;
               x14 : Bool;
               x15 : Bool;
               x00 : Bool;
               x01 : Bool;
               x02 : Bool;
               x03 : Bool;
               x04 : Bool;
               x05 : Bool;
               x06 : Bool;
               x07 : Bool;
            END_STRUCT;
         END_STRUCT;
         speed_ref : Int;
      END_STRUCT;
      write6_stop_mode : Int;
      write7_no_comm_action : Int := 1;   // 1 = Ramp Stop
      c : Int := 1;
      setup_finished : Bool;
   END_VAR
BEGIN
   // Weg - CFW100
   // 
   // Web: http://www.clrwtr.com/PDF/WEG/WEG-CFW100-Programming.pdf

   "mb_station_block_header"(sb := #sb, mb_query := #mb_query);
   #mb_query.mb_addr := #mb_addr;

   #mb_query.mode := #mb_query.c.read.holding_reg;
   #mb_query(data_addr := 2, data_ptr := #read1);
   #mb_query(data_addr := 680, data_ptr := #read2_staus);

   #mb_query.mode := #mb_query.c.write.holding_reg;
   #mb_query(data_addr := 682, data_ptr := #write5);

   #mb_query.Done := false;
   CASE #c OF
       1:
           #mb_query(data_addr := 133, data_ptr := #write1);
       2:
           #mb_query(data_addr := 101, data_ptr := #write2);
       3:
           #mb_query(data_addr := 220, data_ptr := #write3_sel_rem);
       4:
           #mb_query(data_addr := 222, data_ptr := #write4_Ref_sel);
       5:
           #mb_query(data_addr := 229, data_ptr := #write6_stop_mode);
       6:
           #mb_query(data_addr := 313, data_ptr := #write7_no_comm_action);
       ELSE:
           #c := 1;
   END_CASE;
   #c += BOOL_TO_INT(#mb_query.Done);

   "mb_station_block_footer"(sb := #sb, mb_query := #mb_query);
   IF #sb.out.Communication_error THEN
       #setup_finished := false;
   END_IF;

   (*
   P229 Stop mode:
   0 The inverter will apply the stop ramp programmed in P101 or P103.
   1 The motor will run free until it stops

   P006 Inverter Status:
   0 = Ready
   1 = Run
   2 = Undervoltage
   3 = Fault
   4 = Not Used
   5 = Configuration

   *)
END_FUNCTION_BLOCK

FUNCTION_BLOCK "Wika_GDT20_GDHT20"   // FB75, SCL
{ S7_Optimized_Access := 'TRUE' }
VERSION : 0.1
   VAR_INPUT
      mb_addr : UInt;
   END_VAR
   VAR_IN_OUT
      mb_query : "mb_query";
   END_VAR
   VAR
      sb : "mb_station_block_udt";
      data : Struct
         pressure_bar : Real;
         pressure_MPa : Real;
         pressure_Pa : Real;
         pressure_kPa : Real;
         pressure_psi : Real;
         pressure_N_cmÂ² : Real;
         Temperature_C : Real;
         Temperature_K : Real;
         Temperature_F : Real;
         gas_density_g_l : Real;
         gas_density_kg_m3 : Real;
         "Pressure_standardised_to 20_C" : Real;
         Humidity_Atmosphere_frost_point : Real;
         Humidity_Atmosphere_dew_point : Real;
         Humidity_Tank_pressure_frost_point : Real;
         Humidity_Tank_pressure_dew_point_1 : Real;
      END_STRUCT;
      tag : String[16];
      alarm : Struct
         x08_Failure_humidity_sensor : Bool;   // (only model GDHT-20)
         x09_Communication_error_humidity_sensor : Bool;   // (only model GDHT-20)
         x10_Re_occurring_Modbus_communication_error : Bool;   // Re-occurring ModbusÂ® communication error
         x11 : Bool;
         x12 : Bool;
         x13 : Bool;
         x14 : Bool;
         x15 : Bool;
         x00_Pressure_below_lower_limit : Bool;   // Pressure signal below the lower limit value (< 0 bar)
         x01_Pressure_above_upper_limit : Bool;
         x02_Pressure_sensor_failure : Bool;
         x03_Temperature_below_lower_limit : Bool;   // Temperature signal below the lower limit value (< -40 Â°C)
         x04_Temperature_above_upper_limit : Bool;
         x05_Communication_error_pressure_temperature_sensor : Bool;
         x06_Pressure_density_below_lower_limit : Bool;   // Pressure density below the lower limit value (liquefaction of SF6 gas)
         x07_Gas_density_above_upper_limit : Bool;   // Gas density above the upper limit value (> 80 g/l)
      END_STRUCT;
      reset_alarm : Bool;
   END_VAR
   VAR_TEMP
      "int" : Int;
   END_VAR
BEGIN
   // Wika - GDT-20, GDHT-20 (GDT-20, GDHT-20)
   // Pressure / temperature / Gas density / Humidity 
   // 
   // http://en-co.wika.de/upload/OI_GDT_GDHT_20_en_de_67032.pdf

   "mb_station_block_header"(sb := #sb, mb_query := #mb_query);
   #mb_query.mb_addr := #mb_addr;

   #mb_query.mode := #mb_query.c.read.holding_reg;
   #mb_query(data_addr := 0, data_ptr := #data);
   #mb_query(data_addr := 113, data_ptr := #tag);
   #mb_query(data_addr := 200, data_ptr := #alarm);

   IF #reset_alarm THEN
       #"int" := 1;
       #mb_query(mode := #mb_query.c.write.holding_reg,
                 data_addr := 201,
                 data_ptr := #"int");
       IF #mb_query.Done THEN
           #reset_alarm := false;
       END_IF;
   END_IF;

   "mb_station_block_footer"(sb := #sb, mb_query := #mb_query);


   (*
   Circular connector M12 x 1 (5-pin):
   1 C Reference potential RS-485 common
   2 UB Voltage supply (DC 17 ... 30 V)
   3 GND Ground
   4 A Signal RS-485
   5 B Signal RS-485
   *)
END_FUNCTION_BLOCK

// folder: Library/Modbus/Station blocks/sb Untested/Y

FUNCTION_BLOCK "Yaskawa_e7_drive"   // FB76, SCL
{ S7_Optimized_Access := 'TRUE' }
VERSION : 0.1
   VAR_INPUT
      mb_addr : UInt;
   END_VAR
   VAR_IN_OUT
      mb_query : "mb_query";
   END_VAR
   VAR
      sb : "mb_station_block_udt";
      read1 : Struct
         stat : Struct
            x08 : Bool;
            x09 : Bool;
            x10 : Bool;
            x11 : Bool;
            x12 : Bool;
            x13 : Bool;
            x14 : Bool;
            x15 : Bool;
            x00_run : Bool;
            x01 : Bool;
            x02 : Bool;
            x03_reset_signal : Bool;
            x04_speed_agree : Bool;
            x05_inverter_ready : Bool;
            x06_minor_fault : Bool;
            x07_major_fault : Bool;
            "a" : Struct
               x08 : Bool;
               x09 : Bool;
               x10 : Bool;
               x11 : Bool;
               x12 : Bool;
               x13 : Bool;
               x14 : Bool;
               x15 : Bool;
               x00 : Bool;
               x01 : Bool;
               x02 : Bool;
               x03 : Bool;
               x04 : Bool;
               x05 : Bool;
               x06 : Bool;
               x07 : Bool;
            END_STRUCT;
         END_STRUCT;
      END_STRUCT;
      read2 : Struct
         fault_contents_1 : Struct
            x08_inverter_overheat : Bool;
            x09_inverter_overheat_warning : Bool;
            x10_motor_overload : Bool;
            x11_inverter_overload : Bool;
            x12_overtorque_1 : Bool;
            x13_overtorque_2 : Bool;
            x14_braking_resistor_fault : Bool;
            x15_braking_resistor_overheat : Bool;
            x00_fuse : Bool;
            x01_main_circuit_undervoltage : Bool;
            x02_control_circuit_undervoltage : Bool;
            x03_mc_error : Bool;
            x04 : Bool;
            x05_ground_fault : Bool;
            x06_over_current : Bool;
            x07_overvoltage : Bool;
            "a" : Struct
               x08 : Bool;
               x09 : Bool;
               x10 : Bool;
               x11 : Bool;
               x12 : Bool;
               x13 : Bool;
               x14 : Bool;
               x15 : Bool;
               x00 : Bool;
               x01 : Bool;
               x02 : Bool;
               x03 : Bool;
               x04 : Bool;
               x05 : Bool;
               x06 : Bool;
               x07 : Bool;
            END_STRUCT;
         END_STRUCT;
      END_STRUCT;
      read3_data : Struct
         "Output Frequency" : Word;   // 0.01Hz
         "Output Current" : Word;   // 0.1A
         "Output Voltage" : Word;   // 0.1Vac
         "DC Bus Voltage" : Word;   // Vdc
         "Output Power" : Word;   // 0.1kW
      END_STRUCT;
      _ : Bool;
      write1 : Struct
         cmd : Struct
            x08 : Bool;
            x09 : Bool;
            x10 : Bool;
            x11 : Bool;
            x12 : Bool;
            x13 : Bool;
            x14 : Bool;
            x15 : Bool;
            run : Bool := TRUE;   // [00]
            reverse : Bool;   // [01]
            external_fault : Bool;   // [02]
            fault_reset : Bool;   // [03]
            ComNet : Bool := TRUE;   // [04]
            ComCtrl : Bool := TRUE;   // [05]
            x06 : Bool;
            x07 : Bool;
         END_STRUCT;
         freq_ref : Int;
      END_STRUCT;
      write2_max_frequency : UInt := 50;   // 0.1 Hz
      write3 : Struct
         ref_source : Int := 2;   // 0=Operator, 1=Terminals, 2=Serial Com, 3=Option PCB
         run_source : Int := 2;   // 0=Operator, 1=Terminals, 2=Serial Com, 3=Option PCB
         stopp_method : Int := 0;   // 0=Ramp to Stop, 1=Coast to Stop, 2=DCInj to Stop, 3=Coast w/Timer (C1-09)
      END_STRUCT;
   END_VAR
BEGIN
   // Yaskawa - E7 Drive
   // Models: CIMR-E7U* 
   // Web: https://www.ccontrols.com/support/dp/TME711.pdf

   "mb_station_block_header"(sb := #sb, mb_query := #mb_query);
   #mb_query.mb_addr := #mb_addr;

   #mb_query.mode := #mb_query.c.read.holding_reg;
   #mb_query(data_addr := 16#10, data_ptr := #read1);
   #mb_query(data_addr := 16#14, data_ptr := #read2);
   #mb_query(data_addr := 16#41, data_ptr := #read3_data);

   #mb_query.mode := #mb_query.c.write.holding_reg;
   #mb_query(data_addr := 16#303, data_ptr := #write2_max_frequency);
   #mb_query(data_addr := 16#180, data_ptr := #write3);
   #mb_query(data_addr := 16#1, data_ptr := #write1);

   "mb_station_block_footer"(sb := #sb, mb_query := #mb_query);
END_FUNCTION_BLOCK

FUNCTION_BLOCK "Yokogawa_multivariable_transmitter"   // FB77, SCL
{ S7_Optimized_Access := 'TRUE' }
VERSION : 0.1
   VAR_INPUT
      mb_addr : UInt;
   END_VAR
   VAR_IN_OUT
      mb_query : "mb_query";
   END_VAR
   VAR
      sb : "mb_station_block_udt";
      data : Struct
         pres : Real;
         sp : Real;
         et : Real;
      END_STRUCT;
   END_VAR
BEGIN
   // Yokogawa - EJX910A and EJX930A - Multivariable Transmitter
   // web: https://web-material3.yokogawa.com/IM01C25R05-01EN_001.pdf?_ga=
   //      2.43421607.346053457.1505559574-1218156352.1505559574

   "mb_station_block_header"(sb := #sb, mb_query := #mb_query);
   #mb_query.mb_addr := #mb_addr;

   #mb_query(mode := #mb_query.c.read.input_reg,
             data_addr := 401,
             data_ptr := #data);

   "mb_station_block_footer"(sb := #sb, mb_query := #mb_query);
END_FUNCTION_BLOCK

// folder: Library/Modbus/Station blocks/sb Untested/zz Internal special

FUNCTION_BLOCK "temeratur_transmitter"   // FB113, SCL
{ S7_Optimized_Access := 'TRUE' }
VERSION : 0.1
   VAR_OUTPUT
      Temperatur : Real;
   END_VAR
   VAR_IN_OUT
      mb_query : "mb_query";
   END_VAR
   VAR
      sb : "mb_station_block_udt";
   END_VAR
   VAR_TEMP
      tmp : Int;
   END_VAR
BEGIN
   // Temperatur transmitter.

   "mb_station_block_header"(sb := #sb, mb_query := #mb_query);

   #mb_query(mb_addr := 1,
             mode := #mb_query.c.read.holding_reg,
             data_addr := 0,
             data_ptr := #tmp);

   IF #mb_query.Done THEN
       #Temperatur := REAL_TO_INT(#tmp) / 10;
   END_IF;

   "mb_station_block_footer"(sb := #sb, mb_query := #mb_query);
END_FUNCTION_BLOCK